LIN {X 0,Y 383.005,Z 334.275,A -85,B 0,C 180,E1 -11834.306,E2 -11834.306} C_VEL
LIN {X 0,Y 383.071,Z 334.265,A -85,B 0,C 180,E1 -11837.25,E2 -11837.25} C_VEL
LIN {X 0,Y 383.019,Z 334.272,A -85,B 0,C 180,E1 -11840.413,E2 -11840.413} C_VEL
LIN {X 0,Y 383.023,Z 334.273,A -85,B 0,C 180,E1 -11844.045,E2 -11844.045} C_VEL
LIN {X 0,Y 383.002,Z 334.279,A -85,B 0,C 180,E1 -11847.574,E2 -11847.574} C_VEL
LIN {X 0,Y 382.989,Z 334.275,A -85,B 0,C 180,E1 -11850.301,E2 -11850.301} C_VEL
LIN {X 0,Y 383.054,Z 334.267,A -85,B 0,C 180,E1 -11852.699,E2 -11852.699} C_VEL
LIN {X 0,Y 383.049,Z 334.27,A -85,B 0,C 180,E1 -11855.04,E2 -11855.04} C_VEL
LIN {X 0,Y 382.99,Z 334.275,A -85,B 0,C 180,E1 -11858.47,E2 -11858.47} C_VEL
LIN {X 0,Y 383.087,Z 334.264,A -85,B 0,C 180,E1 -11861.828,E2 -11861.828} C_VEL
LIN {X 0,Y 383.108,Z 334.266,A -85,B 0,C 180,E1 -11865.119,E2 -11865.119} C_VEL
LIN {X 0,Y 383.096,Z 334.262,A -85,B 0,C 180,E1 -11868.358,E2 -11868.358} C_VEL
LIN {X 0,Y 383.262,Z 334.241,A -85,B 0,C 180,E1 -11871.977,E2 -11871.977} C_VEL
LIN {X 0,Y 383.196,Z 334.253,A -85,B 0,C 180,E1 -11874.739,E2 -11874.739} C_VEL
LIN {X 0,Y 383.387,Z 334.225,A -85,B 0,C 180,E1 -11877.899,E2 -11877.899} C_VEL
LIN {X 0,Y 383.517,Z 334.209,A -85,B 0,C 180,E1 -11880.001,E2 -11880.001} C_VEL
LIN {X 0,Y 383.249,Z 334.245,A -85,B 0,C 180,E1 -11883.154,E2 -11883.154} C_VEL
LIN {X 0,Y 383.28,Z 334.241,A -85,B 0,C 180,E1 -11886.317,E2 -11886.317} C_VEL
LIN {X 0,Y 383.151,Z 334.254,A -85,B 0,C 180,E1 -11889.503,E2 -11889.503} C_VEL
LIN {X 0,Y 383.125,Z 334.258,A -85,B 0,C 180,E1 -11893.537,E2 -11893.537} C_VEL
LIN {X 0,Y 383.094,Z 334.262,A -85,B 0,C 180,E1 -11897.07,E2 -11897.07} C_VEL
LIN {X 0,Y 383.034,Z 334.272,A -85,B 0,C 180,E1 -11900.65,E2 -11900.65} C_VEL
LIN {X 0,Y 383.023,Z 334.272,A -85,B 0,C 180,E1 -11903.809,E2 -11903.809} C_VEL
LIN {X 0,Y 383.08,Z 334.269,A -85,B 0,C 180,E1 -11906.124,E2 -11906.124} C_VEL
LIN {X 0,Y 383.018,Z 334.274,A -85,B 0,C 180,E1 -11908.495,E2 -11908.495} C_VEL
LIN {X 0,Y 383.011,Z 334.277,A -85,B 0,C 180,E1 -11912.15,E2 -11912.15} C_VEL
LIN {X 0,Y 383.019,Z 334.275,A -85,B 0,C 180,E1 -11914.668,E2 -11914.668} C_VEL
LIN {X 0,Y 383.004,Z 334.279,A -85,B 0,C 180,E1 -11917.905,E2 -11917.905} C_VEL
LIN {X 0,Y 383.462,Z 337.13,A -85,B 0,C 180,E1 -11921.285,E2 -11921.285} C_VEL
LIN {X 0,Y 383.825,Z 340.043,A -85,B 0,C 180,E1 -11924.43,E2 -11924.43} C_VEL
LIN {X 0,Y 384.05,Z 343.012,A -85,B 0,C 180,E1 -11927.384,E2 -11927.384} C_VEL
LIN {X 0,Y 383.867,Z 346.172,A -85,B 0,C 180,E1 -11930.261,E2 -11930.261} C_VEL
LIN {X 0,Y 383.627,Z 349.135,A -85,B 0,C 180,E1 -11932.803,E2 -11932.803} C_VEL
LIN {X 0,Y 383.165,Z 353.821,A -85,B 0,C 180,E1 -11936.615,E2 -11936.615} C_VEL
LIN {X 0,Y 382.799,Z 357.743,A -85,B 0,C 180,E1 -11939.644,E2 -11939.644} C_VEL
LIN {X 0,Y 382.466,Z 361.805,A -85,B 0,C 180,E1 -11942.653,E2 -11942.653} C_VEL
LIN {X 0,Y 382.125,Z 366.674,A -85,B 0,C 180,E1 -11946.133,E2 -11946.133} C_VEL
LIN {X 0,Y 381.861,Z 371.985,A -85,B 0,C 180,E1 -11949.825,E2 -11949.825} C_VEL
LIN {X 0,Y 381.764,Z 373.941,A -85,B 0,C 180,E1 -11951.102,E2 -11951.102} C_VEL
LIN {X 0,Y 383.92,Z 384.326,A -85,B 0,C 180,E1 -11951.558,E2 -11951.558} C_VEL
LIN {X 0,Y 385.496,Z 393.257,A -85,B 0,C 180,E1 -11952.049,E2 -11952.049} C_VEL
LIN {X 0,Y 386.748,Z 402.194,A -85,B 0,C 180,E1 -11952.633,E2 -11952.633} C_VEL
LIN {X 0,Y 387.052,Z 408.906,A -85,B 0,C 180,E1 -11953.111,E2 -11953.111} C_VEL
LIN {X 0,Y 386.18,Z 419.818,A -85,B 0,C 180,E1 -11954.023,E2 -11954.023} C_VEL
LIN {X 0,Y 385.324,Z 428.762,A -85,B 0,C 180,E1 -11954.935,E2 -11954.935} C_VEL
LIN {X 0,Y 384.664,Z 436.503,A -85,B 0,C 180,E1 -11955.879,E2 -11955.879} C_VEL
LIN {X 0,Y 383.999,Z 444.518,A -85,B 0,C 180,E1 -11957.044,E2 -11957.044} C_VEL
LIN {X 0,Y 383.347,Z 450.719,A -85,B 0,C 180,E1 -11958.097,E2 -11958.097} C_VEL
LIN {X 0,Y 382.763,Z 457.257,A -85,B 0,C 180,E1 -11959.42,E2 -11959.42} C_VEL
LIN {X 0,Y 382.4,Z 461.76,A -85,B 0,C 180,E1 -11960.479,E2 -11960.479} C_VEL
LIN {X 0,Y 381.991,Z 467.252,A -85,B 0,C 180,E1 -11962.069,E2 -11962.069} C_VEL
LIN {X 0,Y 381.713,Z 471.576,A -85,B 0,C 180,E1 -11963.658,E2 -11963.658} C_VEL
LIN {X 0,Y 381.646,Z 473.944,A -85,B 0,C 180,E1 -11964.717,E2 -11964.717} C_VEL
LIN {X 0,Y 381.627,Z 475.743,A -85,B 0,C 180,E1 -11965.776,E2 -11965.776} C_VEL
LIN {X 0,Y 381.56,Z 478.187,A -85,B 0,C 180,E1 -11967.889,E2 -11967.889} C_VEL
LIN {X 0,Y 381.603,Z 478.776,A -85,B 0,C 180,E1 -11968.945,E2 -11968.945} C_VEL
LIN {X 0,Y 381.603,Z 478.776,A -85,B 0,C 180,E1 -11971.055,E2 -11971.055} C_VEL
LIN {X 0,Y 381.56,Z 478.187,A -85,B 0,C 180,E1 -11972.111,E2 -11972.111} C_VEL
LIN {X 0,Y 381.627,Z 475.743,A -85,B 0,C 180,E1 -11974.224,E2 -11974.224} C_VEL
LIN {X 0,Y 381.644,Z 473.943,A -85,B 0,C 180,E1 -11975.283,E2 -11975.283} C_VEL
LIN {X 0,Y 381.783,Z 470.336,A -85,B 0,C 180,E1 -11976.872,E2 -11976.872} C_VEL
LIN {X 0,Y 382.116,Z 465.592,A -85,B 0,C 180,E1 -11978.461,E2 -11978.461} C_VEL
LIN {X 0,Y 382.541,Z 459.568,A -85,B 0,C 180,E1 -11980.051,E2 -11980.051} C_VEL
LIN {X 0,Y 383.075,Z 453.471,A -85,B 0,C 180,E1 -11981.375,E2 -11981.375} C_VEL
LIN {X 0,Y 383.666,Z 447.771,A -85,B 0,C 180,E1 -11982.429,E2 -11982.429} C_VEL
LIN {X 0,Y 384.398,Z 439.214,A -85,B 0,C 180,E1 -11983.75,E2 -11983.75} C_VEL
LIN {X 0,Y 385.098,Z 431.032,A -85,B 0,C 180,E1 -11984.803,E2 -11984.803} C_VEL
LIN {X 0,Y 385.884,Z 422.52,A -85,B 0,C 180,E1 -11985.719,E2 -11985.719} C_VEL
LIN {X 0,Y 386.66,Z 413.804,A -85,B 0,C 180,E1 -11986.499,E2 -11986.499} C_VEL
LIN {X 0,Y 387.148,Z 406.33,A -85,B 0,C 180,E1 -11987.07,E2 -11987.07} C_VEL
LIN {X 0,Y 385.973,Z 396.427,A -85,B 0,C 180,E1 -11987.761,E2 -11987.761} C_VEL
LIN {X 0,Y 384.121,Z 385.213,A -85,B 0,C 180,E1 -11988.397,E2 -11988.397} C_VEL
LIN {X 0,Y 381.855,Z 374.444,A -85,B 0,C 180,E1 -11988.88,E2 -11988.88} C_VEL
LIN {X 0,Y 381.785,Z 373.753,A -85,B 0,C 180,E1 -11988.931,E2 -11988.931} C_VEL
LIN {X 0,Y 381.957,Z 369.9,A -85,B 0,C 180,E1 -11991.592,E2 -11991.592} C_VEL
LIN {X 0,Y 382.246,Z 365.004,A -85,B 0,C 180,E1 -11995.016,E2 -11995.016} C_VEL
LIN {X 0,Y 382.585,Z 360.178,A -85,B 0,C 180,E1 -11998.53,E2 -11998.53} C_VEL
LIN {X 0,Y 383.044,Z 355.398,A -85,B 0,C 180,E1 -12002.146,E2 -12002.146} C_VEL
LIN {X 0,Y 383.447,Z 350.679,A -85,B 0,C 180,E1 -12005.91,E2 -12005.91} C_VEL
LIN {X 0,Y 383.765,Z 347.567,A -85,B 0,C 180,E1 -12008.51,E2 -12008.51} C_VEL
LIN {X 0,Y 383.998,Z 344.341,A -85,B 0,C 180,E1 -12011.375,E2 -12011.375} C_VEL
LIN {X 0,Y 383.996,Z 341.509,A -85,B 0,C 180,E1 -12014.066,E2 -12014.066} C_VEL
LIN {X 0,Y 383.581,Z 338.384,A -85,B 0,C 180,E1 -12017.318,E2 -12017.318} C_VEL
LIN {X 0,Y 383.229,Z 335.695,A -85,B 0,C 180,E1 -12020.374,E2 -12020.374} C_VEL
LIN {X 0,Y 383.004,Z 334.279,A -85,B 0,C 180,E1 -12022.095,E2 -12022.095} C_VEL
LIN {X 0,Y 383.019,Z 334.278,A -85,B 0,C 180,E1 -12025.332,E2 -12025.332} C_VEL
LIN {X 0,Y 382.984,Z 334.275,A -85,B 0,C 180,E1 -12029.081,E2 -12029.081} C_VEL
LIN {X 0,Y 383.057,Z 334.266,A -85,B 0,C 180,E1 -12032.698,E2 -12032.698} C_VEL
LIN {X 0,Y 383.051,Z 334.267,A -85,B 0,C 180,E1 -12035.039,E2 -12035.039} C_VEL
LIN {X 0,Y 382.995,Z 334.274,A -85,B 0,C 180,E1 -12038.469,E2 -12038.469} C_VEL
LIN {X 0,Y 383.053,Z 334.271,A -85,B 0,C 180,E1 -12041.825,E2 -12041.825} C_VEL
LIN {X 0,Y 383.11,Z 334.262,A -85,B 0,C 180,E1 -12045.118,E2 -12045.118} C_VEL
LIN {X 0,Y 383.097,Z 334.261,A -85,B 0,C 180,E1 -12048.357,E2 -12048.357} C_VEL
LIN {X 0,Y 383.263,Z 334.241,A -85,B 0,C 180,E1 -12051.975,E2 -12051.975} C_VEL
LIN {X 0,Y 383.196,Z 334.25,A -85,B 0,C 180,E1 -12054.738,E2 -12054.738} C_VEL
LIN {X 0,Y 383.387,Z 334.226,A -85,B 0,C 180,E1 -12057.898,E2 -12057.898} C_VEL
LIN {X 0,Y 383.517,Z 334.209,A -85,B 0,C 180,E1 -12059.999,E2 -12059.999} C_VEL
LIN {X 0,Y 383.25,Z 334.248,A -85,B 0,C 180,E1 -12063.153,E2 -12063.153} C_VEL
LIN {X 0,Y 383.262,Z 334.24,A -85,B 0,C 180,E1 -12066.542,E2 -12066.542} C_VEL
LIN {X 0,Y 383.15,Z 334.256,A -85,B 0,C 180,E1 -12069.502,E2 -12069.502} C_VEL
LIN {X 0,Y 383.123,Z 334.258,A -85,B 0,C 180,E1 -12073.536,E2 -12073.536} C_VEL
LIN {X 0,Y 383.093,Z 334.262,A -85,B 0,C 180,E1 -12077.454,E2 -12077.454} C_VEL
LIN {X 0,Y 383.027,Z 334.276,A -85,B 0,C 180,E1 -12080.646,E2 -12080.646} C_VEL
LIN {X 0,Y 383.023,Z 334.271,A -85,B 0,C 180,E1 -12083.807,E2 -12083.807} C_VEL
LIN {X 0,Y 383.077,Z 334.266,A -85,B 0,C 180,E1 -12086.123,E2 -12086.123} C_VEL
LIN {X 0,Y 383.037,Z 334.275,A -85,B 0,C 180,E1 -12088.492,E2 -12088.492} C_VEL
LIN {X 0,Y 383.006,Z 334.276,A -85,B 0,C 180,E1 -12092.149,E2 -12092.149} C_VEL
LIN {X 0,Y 383.015,Z 334.274,A -85,B 0,C 180,E1 -12094.667,E2 -12094.667} C_VEL
LIN {X 0,Y 383,Z 334.276,A -85,B 0,C 180,E1 -12097.904,E2 -12097.904} C_VEL
LIN {X 0,Y 383.043,Z 334.268,A -85,B 0,C 180,E1 -12101.339,E2 -12101.339} C_VEL
LIN {X 0,Y 383.033,Z 334.273,A -85,B 0,C 180,E1 -12104.309,E2 -12104.309} C_VEL
LIN {X 0,Y 383.036,Z 334.269,A -85,B 0,C 180,E1 -12107.244,E2 -12107.244} C_VEL
LIN {X 0,Y 383.018,Z 334.273,A -85,B 0,C 180,E1 -12110.412,E2 -12110.412} C_VEL
LIN {X 0,Y 383.023,Z 334.275,A -85,B 0,C 180,E1 -12114.044,E2 -12114.044} C_VEL
LIN {X 0,Y 382.983,Z 334.28,A -85,B 0,C 180,E1 -12117.578,E2 -12117.578} C_VEL
LIN {X 0,Y 382.988,Z 334.276,A -85,B 0,C 180,E1 -12120.3,E2 -12120.3} C_VEL
LIN {X 0,Y 383.053,Z 334.267,A -85,B 0,C 180,E1 -12122.698,E2 -12122.698} C_VEL
LIN {X 0,Y 383.03,Z 334.27,A -85,B 0,C 180,E1 -12126.193,E2 -12126.193} C_VEL
LIN {X 0,Y 383.056,Z 334.272,A -85,B 0,C 180,E1 -12129.599,E2 -12129.599} C_VEL
LIN {X 0,Y 383.101,Z 334.266,A -85,B 0,C 180,E1 -12132.931,E2 -12132.931} C_VEL
LIN {X 0,Y 383.121,Z 334.263,A -85,B 0,C 180,E1 -12136.464,E2 -12136.464} C_VEL
LIN {X 0,Y 383.139,Z 334.266,A -85,B 0,C 180,E1 -12139.597,E2 -12139.597} C_VEL
LIN {X 0,Y 383.738,Z 336.384,A -85,B 0,C 180,E1 -12139.914,E2 -12139.914} C_VEL
LIN {X 0,Y 385.2,Z 338.424,A -85,B 0,C 180,E1 -12140.615,E2 -12140.615} C_VEL
LIN {X 0,Y 387.437,Z 339.864,A -85,B 0,C 180,E1 -12141.656,E2 -12141.656} C_VEL
LIN {X 0,Y 388.84,Z 340.559,A -85,B 0,C 180,E1 -12142.402,E2 -12142.402} C_VEL
LIN {X 0,Y 389.961,Z 342.834,A -85,B 0,C 180,E1 -12143.142,E2 -12143.142} C_VEL
LIN {X 0,Y 391.789,Z 344.996,A -85,B 0,C 180,E1 -12144.467,E2 -12144.467} C_VEL
LIN {X 0,Y 393.422,Z 346.061,A -85,B 0,C 180,E1 -12145.902,E2 -12145.902} C_VEL
LIN {X 0,Y 394.945,Z 346.431,A -85,B 0,C 180,E1 -12147.96,E2 -12147.96} C_VEL
LIN {X 0,Y 395.509,Z 346.494,A -85,B 0,C 180,E1 -12150,E2 -12150} C_VEL
LIN {X 0,Y 394.945,Z 346.431,A -85,B 0,C 180,E1 -12152.04,E2 -12152.04} C_VEL
LIN {X 0,Y 393.422,Z 346.062,A -85,B 0,C 180,E1 -12154.098,E2 -12154.098} C_VEL
LIN {X 0,Y 391.445,Z 344.701,A -85,B 0,C 180,E1 -12155.796,E2 -12155.796} C_VEL
LIN {X 0,Y 389.552,Z 342.156,A -85,B 0,C 180,E1 -12157.135,E2 -12157.135} C_VEL
LIN {X 0,Y 388.788,Z 340.393,A -85,B 0,C 180,E1 -12157.634,E2 -12157.634} C_VEL
LIN {X 0,Y 385.957,Z 339.051,A -85,B 0,C 180,E1 -12159.036,E2 -12159.036} C_VEL
LIN {X 0,Y 384.054,Z 336.971,A -85,B 0,C 180,E1 -12159.938,E2 -12159.938} C_VEL
LIN {X 0,Y 383.252,Z 334.909,A -85,B 0,C 180,E1 -12160.333,E2 -12160.333} C_VEL
LIN {X 0,Y 383.121,Z 334.263,A -85,B 0,C 180,E1 -12160.436,E2 -12160.436} C_VEL
LIN {X 0,Y 383.123,Z 334.262,A -85,B 0,C 180,E1 -12163.796,E2 -12163.796} C_VEL
LIN {X 0,Y 383.091,Z 334.266,A -85,B 0,C 180,E1 -12167.455,E2 -12167.455} C_VEL
LIN {X 0,Y 383.03,Z 334.274,A -85,B 0,C 180,E1 -12170.649,E2 -12170.649} C_VEL
LIN {X 0,Y 383.03,Z 334.27,A -85,B 0,C 180,E1 -12173.807,E2 -12173.807} C_VEL
LIN {X 0,Y 383.053,Z 334.267,A -85,B 0,C 180,E1 -12177.302,E2 -12177.302} C_VEL
LIN {X 0,Y 382.979,Z 334.277,A -85,B 0,C 180,E1 -12180.919,E2 -12180.919} C_VEL
LIN {X 0,Y 383.014,Z 334.273,A -85,B 0,C 180,E1 -12184.668,E2 -12184.668} C_VEL
LIN {X 0,Y 382.995,Z 334.274,A -85,B 0,C 180,E1 -12185.364,E2 -12185.364} C_VEL
LIN {X 0,Y 382.354,Z 334.359,A -85,B 0,C 180,E1 -12186.242,E2 -12186.242} C_VEL
LIN {X 0,Y 379.547,Z 334.716,A -85,B 0,C 180,E1 -12187.67,E2 -12187.67} C_VEL
LIN {X 0,Y 377.144,Z 335.017,A -85,B 0,C 180,E1 -12188.824,E2 -12188.824} C_VEL
LIN {X 0,Y 376.089,Z 335.143,A -85,B 0,C 180,E1 -12189.716,E2 -12189.716} C_VEL
LIN {X 0,Y 375.991,Z 335.152,A -85,B 0,C 180,E1 -12190.019,E2 -12190.019} C_VEL
LIN {X 0,Y 375.943,Z 335.157,A -85,B 0,C 180,E1 -12193.764,E2 -12193.764} C_VEL
LIN {X 0,Y 375.986,Z 335.147,A -85,B 0,C 180,E1 -12196.802,E2 -12196.802} C_VEL
LIN {X 0,Y 375.996,Z 335.15,A -85,B 0,C 180,E1 -12200.028,E2 -12200.028} C_VEL
LIN {X 0,Y 375.962,Z 335.154,A -85,B 0,C 180,E1 -12203.496,E2 -12203.496} C_VEL
LIN {X 0,Y 375.957,Z 335.154,A -85,B 0,C 180,E1 -12205.889,E2 -12205.889} C_VEL
LIN {X 0,Y 375.961,Z 335.155,A -85,B 0,C 180,E1 -12209.688,E2 -12209.688} C_VEL
LIN {X 0,Y 375.993,Z 335.147,A -85,B 0,C 180,E1 -12212.142,E2 -12212.142} C_VEL
LIN {X 0,Y 376.003,Z 335.145,A -85,B 0,C 180,E1 -12214.539,E2 -12214.539} C_VEL
LIN {X 0,Y 375.956,Z 335.151,A -85,B 0,C 180,E1 -12218.046,E2 -12218.046} C_VEL
LIN {X 0,Y 376.022,Z 335.147,A -85,B 0,C 180,E1 -12221.475,E2 -12221.475} C_VEL
LIN {X 0,Y 376.056,Z 335.141,A -85,B 0,C 180,E1 -12224.833,E2 -12224.833} C_VEL
LIN {X 0,Y 376.048,Z 335.139,A -85,B 0,C 180,E1 -12228.137,E2 -12228.137} C_VEL
LIN {X 0,Y 376.217,Z 335.118,A -85,B 0,C 180,E1 -12231.92,E2 -12231.92} C_VEL
LIN {X 0,Y 376.168,Z 335.127,A -85,B 0,C 180,E1 -12234.64,E2 -12234.64} C_VEL
LIN {X 0,Y 376.353,Z 335.101,A -85,B 0,C 180,E1 -12237.86,E2 -12237.86} C_VEL
LIN {X 0,Y 376.486,Z 335.085,A -85,B 0,C 180,E1 -12240.001,E2 -12240.001} C_VEL
LIN {X 0,Y 376.187,Z 335.124,A -85,B 0,C 180,E1 -12243.213,E2 -12243.213} C_VEL
LIN {X 0,Y 376.238,Z 335.12,A -85,B 0,C 180,E1 -12246.436,E2 -12246.436} C_VEL
LIN {X 0,Y 376.119,Z 335.13,A -85,B 0,C 180,E1 -12249.682,E2 -12249.682} C_VEL
LIN {X 0,Y 376.089,Z 335.134,A -85,B 0,C 180,E1 -12253.658,E2 -12253.658} C_VEL
LIN {X 0,Y 376.032,Z 335.141,A -85,B 0,C 180,E1 -12257.4,E2 -12257.4} C_VEL
LIN {X 0,Y 375.978,Z 335.149,A -85,B 0,C 180,E1 -12260.833,E2 -12260.833} C_VEL
LIN {X 0,Y 375.988,Z 335.153,A -85,B 0,C 180,E1 -12264.282,E2 -12264.282} C_VEL
LIN {X 0,Y 376.02,Z 335.145,A -85,B 0,C 180,E1 -12266.653,E2 -12266.653} C_VEL
LIN {X 0,Y 375.965,Z 335.154,A -85,B 0,C 180,E1 -12270.313,E2 -12270.313} C_VEL
LIN {X 0,Y 375.961,Z 335.157,A -85,B 0,C 180,E1 -12274.112,E2 -12274.112} C_VEL
LIN {X 0,Y 375.955,Z 335.156,A -85,B 0,C 180,E1 -12276.742,E2 -12276.742} C_VEL
LIN {X 0,Y 376.033,Z 335.725,A -85,B 0,C 180,E1 -12278.282,E2 -12278.282} C_VEL
LIN {X 0,Y 376.483,Z 338.576,A -85,B 0,C 180,E1 -12281.695,E2 -12281.695} C_VEL
LIN {X 0,Y 376.879,Z 341.755,A -85,B 0,C 180,E1 -12285.123,E2 -12285.123} C_VEL
LIN {X 0,Y 376.982,Z 344.5,A -85,B 0,C 180,E1 -12287.845,E2 -12287.845} C_VEL
LIN {X 0,Y 376.792,Z 347.545,A -85,B 0,C 180,E1 -12290.641,E2 -12290.641} C_VEL
LIN {X 0,Y 376.515,Z 350.697,A -85,B 0,C 180,E1 -12293.383,E2 -12293.383} C_VEL
LIN {X 0,Y 376.027,Z 355.41,A -85,B 0,C 180,E1 -12297.253,E2 -12297.253} C_VEL
LIN {X 0,Y 375.744,Z 358.488,A -85,B 0,C 180,E1 -12299.668,E2 -12299.668} C_VEL
LIN {X 0,Y 375.313,Z 363.296,A -85,B 0,C 180,E1 -12303.294,E2 -12303.294} C_VEL
LIN {X 0,Y 375.014,Z 368.142,A -85,B 0,C 180,E1 -12306.824,E2 -12306.824} C_VEL
LIN {X 0,Y 374.741,Z 373.736,A -85,B 0,C 180,E1 -12310.734,E2 -12310.734} C_VEL
LIN {X 0,Y 376.765,Z 383.476,A -85,B 0,C 180,E1 -12311.169,E2 -12311.169} C_VEL
LIN {X 0,Y 378.478,Z 393.112,A -85,B 0,C 180,E1 -12311.708,E2 -12311.708} C_VEL
LIN {X 0,Y 379.829,Z 402.363,A -85,B 0,C 180,E1 -12312.332,E2 -12312.332} C_VEL
LIN {X 0,Y 380.242,Z 408.71,A -85,B 0,C 180,E1 -12312.799,E2 -12312.799} C_VEL
LIN {X 0,Y 379.337,Z 419.622,A -85,B 0,C 180,E1 -12313.727,E2 -12313.727} C_VEL
LIN {X 0,Y 378.449,Z 428.566,A -85,B 0,C 180,E1 -12314.655,E2 -12314.655} C_VEL
LIN {X 0,Y 377.606,Z 437.835,A -85,B 0,C 180,E1 -12315.829,E2 -12315.829} C_VEL
LIN {X 0,Y 376.887,Z 445.948,A -85,B 0,C 180,E1 -12317.07,E2 -12317.07} C_VEL
LIN {X 0,Y 376.219,Z 451.898,A -85,B 0,C 180,E1 -12318.142,E2 -12318.142} C_VEL
LIN {X 0,Y 375.658,Z 458.217,A -85,B 0,C 180,E1 -12319.49,E2 -12319.49} C_VEL
LIN {X 0,Y 375.215,Z 463.48,A -85,B 0,C 180,E1 -12320.839,E2 -12320.839} C_VEL
LIN {X 0,Y 374.809,Z 468.609,A -85,B 0,C 180,E1 -12322.458,E2 -12322.458} C_VEL
LIN {X 0,Y 374.586,Z 472.267,A -85,B 0,C 180,E1 -12323.931,E2 -12323.931} C_VEL
LIN {X 0,Y 374.553,Z 475.547,A -85,B 0,C 180,E1 -12325.696,E2 -12325.696} C_VEL
LIN {X 0,Y 374.459,Z 477.991,A -85,B 0,C 180,E1 -12327.849,E2 -12327.849} C_VEL
LIN {X 0,Y 374.503,Z 478.581,A -85,B 0,C 180,E1 -12328.925,E2 -12328.925} C_VEL
LIN {X 0,Y 374.503,Z 478.581,A -85,B 0,C 180,E1 -12331.075,E2 -12331.075} C_VEL
LIN {X 0,Y 374.459,Z 477.991,A -85,B 0,C 180,E1 -12332.151,E2 -12332.151} C_VEL
LIN {X 0,Y 374.553,Z 475.547,A -85,B 0,C 180,E1 -12334.304,E2 -12334.304} C_VEL
LIN {X 0,Y 374.584,Z 472.274,A -85,B 0,C 180,E1 -12336.066,E2 -12336.066} C_VEL
LIN {X 0,Y 374.809,Z 468.609,A -85,B 0,C 180,E1 -12337.542,E2 -12337.542} C_VEL
LIN {X 0,Y 375.215,Z 463.48,A -85,B 0,C 180,E1 -12339.161,E2 -12339.161} C_VEL
LIN {X 0,Y 375.657,Z 458.217,A -85,B 0,C 180,E1 -12340.51,E2 -12340.51} C_VEL
LIN {X 0,Y 376.221,Z 451.898,A -85,B 0,C 180,E1 -12341.858,E2 -12341.858} C_VEL
LIN {X 0,Y 376.888,Z 445.948,A -85,B 0,C 180,E1 -12342.93,E2 -12342.93} C_VEL
LIN {X 0,Y 377.606,Z 437.829,A -85,B 0,C 180,E1 -12344.172,E2 -12344.172} C_VEL
LIN {X 0,Y 378.312,Z 429.7,A -85,B 0,C 180,E1 -12345.213,E2 -12345.213} C_VEL
LIN {X 0,Y 379.163,Z 420.972,A -85,B 0,C 180,E1 -12346.143,E2 -12346.143} C_VEL
LIN {X 0,Y 379.955,Z 411.975,A -85,B 0,C 180,E1 -12346.937,E2 -12346.937} C_VEL
LIN {X 0,Y 380.215,Z 406.272,A -85,B 0,C 180,E1 -12347.382,E2 -12347.382} C_VEL
LIN {X 0,Y 378.828,Z 395.108,A -85,B 0,C 180,E1 -12348.167,E2 -12348.167} C_VEL
LIN {X 0,Y 376.872,Z 384.021,A -85,B 0,C 180,E1 -12348.803,E2 -12348.803} C_VEL
LIN {X 0,Y 374.76,Z 373.587,A -85,B 0,C 180,E1 -12349.3,E2 -12349.3} C_VEL
LIN {X 0,Y 375.022,Z 367.931,A -85,B 0,C 180,E1 -12353.324,E2 -12353.324} C_VEL
LIN {X 0,Y 375.314,Z 363.287,A -85,B 0,C 180,E1 -12356.706,E2 -12356.706} C_VEL
LIN {X 0,Y 375.745,Z 358.481,A -85,B 0,C 180,E1 -12360.332,E2 -12360.332} C_VEL
LIN {X 0,Y 376.172,Z 353.737,A -85,B 0,C 180,E1 -12364.089,E2 -12364.089} C_VEL
LIN {X 0,Y 376.66,Z 349.076,A -85,B 0,C 180,E1 -12368.005,E2 -12368.005} C_VEL
LIN {X 0,Y 376.915,Z 346.003,A -85,B 0,C 180,E1 -12370.739,E2 -12370.739} C_VEL
LIN {X 0,Y 376.992,Z 342.998,A -85,B 0,C 180,E1 -12373.611,E2 -12373.611} C_VEL
LIN {X 0,Y 376.651,Z 340.041,A -85,B 0,C 180,E1 -12376.694,E2 -12376.694} C_VEL
LIN {X 0,Y 376.265,Z 337.155,A -85,B 0,C 180,E1 -12379.979,E2 -12379.979} C_VEL
LIN {X 0,Y 376.012,Z 335.567,A -85,B 0,C 180,E1 -12381.917,E2 -12381.917} C_VEL
LIN {X 0,Y 375.965,Z 335.155,A -85,B 0,C 180,E1 -12383.495,E2 -12383.495} C_VEL
LIN {X 0,Y 375.961,Z 335.157,A -85,B 0,C 180,E1 -12385.888,E2 -12385.888} C_VEL
LIN {X 0,Y 375.965,Z 335.154,A -85,B 0,C 180,E1 -12389.687,E2 -12389.687} C_VEL
LIN {X 0,Y 376.02,Z 335.145,A -85,B 0,C 180,E1 -12393.347,E2 -12393.347} C_VEL
LIN {X 0,Y 375.979,Z 335.148,A -85,B 0,C 180,E1 -12396.887,E2 -12396.887} C_VEL
LIN {X 0,Y 375.999,Z 335.146,A -85,B 0,C 180,E1 -12400.339,E2 -12400.339} C_VEL
LIN {X 0,Y 376.026,Z 335.147,A -85,B 0,C 180,E1 -12403.718,E2 -12403.718} C_VEL
LIN {X 0,Y 376.103,Z 335.134,A -85,B 0,C 180,E1 -12407.041,E2 -12407.041} C_VEL
LIN {X 0,Y 376.119,Z 335.13,A -85,B 0,C 180,E1 -12410.318,E2 -12410.318} C_VEL
LIN {X 0,Y 376.238,Z 335.12,A -85,B 0,C 180,E1 -12413.564,E2 -12413.564} C_VEL
LIN {X 0,Y 376.353,Z 335.102,A -85,B 0,C 180,E1 -12417.859,E2 -12417.859} C_VEL
LIN {X 0,Y 376.486,Z 335.085,A -85,B 0,C 180,E1 -12419.999,E2 -12419.999} C_VEL
LIN {X 0,Y 376.188,Z 335.127,A -85,B 0,C 180,E1 -12423.212,E2 -12423.212} C_VEL
LIN {X 0,Y 376.229,Z 335.117,A -85,B 0,C 180,E1 -12426.529,E2 -12426.529} C_VEL
LIN {X 0,Y 376.118,Z 335.131,A -85,B 0,C 180,E1 -12429.681,E2 -12429.681} C_VEL
LIN {X 0,Y 376.088,Z 335.135,A -85,B 0,C 180,E1 -12433.657,E2 -12433.657} C_VEL
LIN {X 0,Y 376.042,Z 335.14,A -85,B 0,C 180,E1 -12437.607,E2 -12437.607} C_VEL
LIN {X 0,Y 375.976,Z 335.153,A -85,B 0,C 180,E1 -12440.832,E2 -12440.832} C_VEL
LIN {X 0,Y 375.987,Z 335.15,A -85,B 0,C 180,E1 -12444.281,E2 -12444.281} C_VEL
LIN {X 0,Y 376.017,Z 335.148,A -85,B 0,C 180,E1 -12446.652,E2 -12446.652} C_VEL
LIN {X 0,Y 375.967,Z 335.15,A -85,B 0,C 180,E1 -12449.079,E2 -12449.079} C_VEL
LIN {X 0,Y 375.953,Z 335.153,A -85,B 0,C 180,E1 -12452.827,E2 -12452.827} C_VEL
LIN {X 0,Y 375.955,Z 335.151,A -85,B 0,C 180,E1 -12455.415,E2 -12455.415} C_VEL
LIN {X 0,Y 375.974,Z 335.155,A -85,B 0,C 180,E1 -12458.271,E2 -12458.271} C_VEL
LIN {X 0,Y 375.986,Z 335.148,A -85,B 0,C 180,E1 -12461.61,E2 -12461.61} C_VEL
LIN {X 0,Y 375.967,Z 335.15,A -85,B 0,C 180,E1 -12465.262,E2 -12465.262} C_VEL
LIN {X 0,Y 375.977,Z 335.148,A -85,B 0,C 180,E1 -12469.138,E2 -12469.138} C_VEL
LIN {X 0,Y 375.964,Z 335.156,A -85,B 0,C 180,E1 -12471.912,E2 -12471.912} C_VEL
LIN {X 0,Y 375.976,Z 335.15,A -85,B 0,C 180,E1 -12475.332,E2 -12475.332} C_VEL
LIN {X 0,Y 375.954,Z 335.152,A -85,B 0,C 180,E1 -12478.438,E2 -12478.438} C_VEL
LIN {X 0,Y 375.992,Z 335.148,A -85,B 0,C 180,E1 -12482.141,E2 -12482.141} C_VEL
LIN {X 0,Y 376.002,Z 335.145,A -85,B 0,C 180,E1 -12484.539,E2 -12484.539} C_VEL
LIN {X 0,Y 375.961,Z 335.152,A -85,B 0,C 180,E1 -12488.046,E2 -12488.046} C_VEL
LIN {X 0,Y 376.021,Z 335.149,A -85,B 0,C 180,E1 -12491.474,E2 -12491.474} C_VEL
LIN {X 0,Y 376.055,Z 335.144,A -85,B 0,C 180,E1 -12494.833,E2 -12494.833} C_VEL
LIN {X 0,Y 376.117,Z 335.308,A -85,B 0,C 180,E1 -12497.317,E2 -12497.317} C_VEL
LIN {X 0,Y 376.775,Z 337.476,A -85,B 0,C 180,E1 -12497.613,E2 -12497.613} C_VEL
LIN {X 0,Y 378.603,Z 339.764,A -85,B 0,C 180,E1 -12498.286,E2 -12498.286} C_VEL
LIN {X 0,Y 381.129,Z 341.2,A -85,B 0,C 180,E1 -12499.206,E2 -12499.206} C_VEL
LIN {X 0,Y 382.563,Z 343.884,A -85,B 0,C 180,E1 -12499.849,E2 -12499.849} C_VEL
LIN {X 0,Y 384.983,Z 346.162,A -85,B 0,C 180,E1 -12500.941,E2 -12500.941} C_VEL
LIN {X 0,Y 387.406,Z 347.441,A -85,B 0,C 180,E1 -12502.125,E2 -12502.125} C_VEL
LIN {X 0,Y 388.935,Z 349.999,A -85,B 0,C 180,E1 -12503.079,E2 -12503.079} C_VEL
LIN {X 0,Y 390.889,Z 352.078,A -85,B 0,C 180,E1 -12504.454,E2 -12504.454} C_VEL
LIN {X 0,Y 392.534,Z 353.091,A -85,B 0,C 180,E1 -12505.893,E2 -12505.893} C_VEL
LIN {X 0,Y 394.083,Z 353.478,A -85,B 0,C 180,E1 -12507.956,E2 -12507.956} C_VEL
LIN {X 0,Y 394.645,Z 353.533,A -85,B 0,C 180,E1 -12510,E2 -12510} C_VEL
LIN {X 0,Y 394.082,Z 353.477,A -85,B 0,C 180,E1 -12512.044,E2 -12512.044} C_VEL
LIN {X 0,Y 392.534,Z 353.092,A -85,B 0,C 180,E1 -12514.107,E2 -12514.107} C_VEL
LIN {X 0,Y 390.528,Z 351.798,A -85,B 0,C 180,E1 -12515.81,E2 -12515.81} C_VEL
LIN {X 0,Y 388.395,Z 349.209,A -85,B 0,C 180,E1 -12517.277,E2 -12517.277} C_VEL
LIN {X 0,Y 387.179,Z 347.137,A -85,B 0,C 180,E1 -12518.008,E2 -12518.008} C_VEL
LIN {X 0,Y 384.526,Z 345.833,A -85,B 0,C 180,E1 -12519.267,E2 -12519.267} C_VEL
LIN {X 0,Y 382.398,Z 343.659,A -85,B 0,C 180,E1 -12520.222,E2 -12520.222} C_VEL
LIN {X 0,Y 380.993,Z 341.031,A -85,B 0,C 180,E1 -12520.852,E2 -12520.852} C_VEL
LIN {X 0,Y 378.582,Z 339.746,A -85,B 0,C 180,E1 -12521.722,E2 -12521.722} C_VEL
LIN {X 0,Y 376.775,Z 337.476,A -85,B 0,C 180,E1 -12522.387,E2 -12522.387} C_VEL
LIN {X 0,Y 376.109,Z 335.138,A -85,B 0,C 180,E1 -12522.718,E2 -12522.718} C_VEL
LIN {X 0,Y 376.025,Z 335.147,A -85,B 0,C 180,E1 -12526.281,E2 -12526.281} C_VEL
LIN {X 0,Y 375.996,Z 335.148,A -85,B 0,C 180,E1 -12529.661,E2 -12529.661} C_VEL
LIN {X 0,Y 375.992,Z 335.147,A -85,B 0,C 180,E1 -12533.668,E2 -12533.668} C_VEL
LIN {X 0,Y 376.016,Z 335.147,A -85,B 0,C 180,E1 -12536.652,E2 -12536.652} C_VEL
LIN {X 0,Y 375.966,Z 335.15,A -85,B 0,C 180,E1 -12539.079,E2 -12539.079} C_VEL
LIN {X 0,Y 375.947,Z 335.153,A -85,B 0,C 180,E1 -12542.829,E2 -12542.829} C_VEL
LIN {X 0,Y 375.955,Z 335.151,A -85,B 0,C 180,E1 -12545.416,E2 -12545.416} C_VEL
LIN {X 0,Y 375.974,Z 335.153,A -85,B 0,C 180,E1 -12548.271,E2 -12548.271} C_VEL
LIN {X 0,Y 375.991,Z 335.152,A -85,B 0,C 180,E1 -12550.019,E2 -12550.019} C_VEL
LIN {X 0,Y 375.278,Z 335.235,A -85,B 0,C 180,E1 -12550.912,E2 -12550.912} C_VEL
LIN {X 0,Y 372.374,Z 335.599,A -85,B 0,C 180,E1 -12552.364,E2 -12552.364} C_VEL
LIN {X 0,Y 369.966,Z 335.899,A -85,B 0,C 180,E1 -12553.539,E2 -12553.539} C_VEL
LIN {X 0,Y 368.975,Z 336.022,A -85,B 0,C 180,E1 -12554.447,E2 -12554.447} C_VEL
LIN {X 0,Y 368.916,Z 336.027,A -85,B 0,C 180,E1 -12554.755,E2 -12554.755} C_VEL
LIN {X 0,Y 368.942,Z 336.027,A -85,B 0,C 180,E1 -12558.187,E2 -12558.187} C_VEL
LIN {X 0,Y 368.909,Z 336.031,A -85,B 0,C 180,E1 -12561.359,E2 -12561.359} C_VEL
LIN {X 0,Y 368.933,Z 336.027,A -85,B 0,C 180,E1 -12565.147,E2 -12565.147} C_VEL
LIN {X 0,Y 368.926,Z 336.028,A -85,B 0,C 180,E1 -12569.047,E2 -12569.047} C_VEL
LIN {X 0,Y 368.977,Z 336.026,A -85,B 0,C 180,E1 -12571.564,E2 -12571.564} C_VEL
LIN {X 0,Y 368.997,Z 336.019,A -85,B 0,C 180,E1 -12574.02,E2 -12574.02} C_VEL
LIN {X 0,Y 368.923,Z 336.031,A -85,B 0,C 180,E1 -12577.605,E2 -12577.605} C_VEL
LIN {X 0,Y 368.98,Z 336.024,A -85,B 0,C 180,E1 -12581.108,E2 -12581.108} C_VEL
LIN {X 0,Y 368.996,Z 336.018,A -85,B 0,C 180,E1 -12584.536,E2 -12584.536} C_VEL
LIN {X 0,Y 369.003,Z 336.017,A -85,B 0,C 180,E1 -12587.907,E2 -12587.907} C_VEL
LIN {X 0,Y 369.186,Z 335.994,A -85,B 0,C 180,E1 -12591.847,E2 -12591.847} C_VEL
LIN {X 0,Y 369.141,Z 336.002,A -85,B 0,C 180,E1 -12594.538,E2 -12594.538} C_VEL
LIN {X 0,Y 369.318,Z 335.978,A -85,B 0,C 180,E1 -12597.819,E2 -12597.819} C_VEL
LIN {X 0,Y 369.456,Z 335.961,A -85,B 0,C 180,E1 -12600.001,E2 -12600.001} C_VEL
LIN {X 0,Y 369.318,Z 335.979,A -85,B 0,C 180,E1 -12602.182,E2 -12602.182} C_VEL
LIN {X 0,Y 369.198,Z 335.998,A -85,B 0,C 180,E1 -12606.559,E2 -12606.559} C_VEL
LIN {X 0,Y 369.121,Z 336.007,A -85,B 0,C 180,E1 -12608.762,E2 -12608.762} C_VEL
LIN {X 0,Y 369.005,Z 336.019,A -85,B 0,C 180,E1 -12612.094,E2 -12612.094} C_VEL
LIN {X 0,Y 368.997,Z 336.018,A -85,B 0,C 180,E1 -12615.465,E2 -12615.465} C_VEL
LIN {X 0,Y 368.955,Z 336.024,A -85,B 0,C 180,E1 -12618.895,E2 -12618.895} C_VEL
LIN {X 0,Y 368.924,Z 336.032,A -85,B 0,C 180,E1 -12622.396,E2 -12622.396} C_VEL
LIN {X 0,Y 369,Z 336.021,A -85,B 0,C 180,E1 -12625.981,E2 -12625.981} C_VEL
LIN {X 0,Y 368.915,Z 336.03,A -85,B 0,C 180,E1 -12629.691,E2 -12629.691} C_VEL
LIN {X 0,Y 368.898,Z 336.03,A -85,B 0,C 180,E1 -12633.044,E2 -12633.044} C_VEL
LIN {X 0,Y 368.918,Z 336.034,A -85,B 0,C 180,E1 -12636.197,E2 -12636.197} C_VEL
LIN {X 0,Y 368.946,Z 336.298,A -85,B 0,C 180,E1 -12637.559,E2 -12637.559} C_VEL
LIN {X 0,Y 369.31,Z 338.591,A -85,B 0,C 180,E1 -12640.43,E2 -12640.43} C_VEL
LIN {X 0,Y 369.701,Z 341.519,A -85,B 0,C 180,E1 -12643.749,E2 -12643.749} C_VEL
LIN {X 0,Y 369.972,Z 344.487,A -85,B 0,C 180,E1 -12646.854,E2 -12646.854} C_VEL
LIN {X 0,Y 369.816,Z 347.5,A -85,B 0,C 180,E1 -12649.749,E2 -12649.749} C_VEL
LIN {X 0,Y 369.513,Z 351.141,A -85,B 0,C 180,E1 -12653.019,E2 -12653.019} C_VEL
LIN {X 0,Y 369.054,Z 355.237,A -85,B 0,C 180,E1 -12656.478,E2 -12656.478} C_VEL
LIN {X 0,Y 368.754,Z 358.424,A -85,B 0,C 180,E1 -12659.054,E2 -12659.054} C_VEL
LIN {X 0,Y 368.295,Z 363.168,A -85,B 0,C 180,E1 -12662.743,E2 -12662.743} C_VEL
LIN {X 0,Y 367.959,Z 368.151,A -85,B 0,C 180,E1 -12666.464,E2 -12666.464} C_VEL
LIN {X 0,Y 367.658,Z 373.51,A -85,B 0,C 180,E1 -12670.348,E2 -12670.348} C_VEL
LIN {X 0,Y 369.811,Z 383.807,A -85,B 0,C 180,E1 -12670.823,E2 -12670.823} C_VEL
LIN {X 0,Y 371.532,Z 393.17,A -85,B 0,C 180,E1 -12671.368,E2 -12671.368} C_VEL
LIN {X 0,Y 372.845,Z 402.504,A -85,B 0,C 180,E1 -12672.014,E2 -12672.014} C_VEL
LIN {X 0,Y 373.408,Z 408.512,A -85,B 0,C 180,E1 -12672.474,E2 -12672.474} C_VEL
LIN {X 0,Y 372.514,Z 419.425,A -85,B 0,C 180,E1 -12673.42,E2 -12673.42} C_VEL
LIN {X 0,Y 371.598,Z 428.37,A -85,B 0,C 180,E1 -12674.365,E2 -12674.365} C_VEL
LIN {X 0,Y 370.905,Z 435.609,A -85,B 0,C 180,E1 -12675.271,E2 -12675.271} C_VEL
LIN {X 0,Y 370.133,Z 444.125,A -85,B 0,C 180,E1 -12676.55,E2 -12676.55} C_VEL
LIN {X 0,Y 369.441,Z 450.326,A -85,B 0,C 180,E1 -12677.642,E2 -12677.642} C_VEL
LIN {X 0,Y 368.725,Z 456.863,A -85,B 0,C 180,E1 -12679.012,E2 -12679.012} C_VEL
LIN {X 0,Y 368.314,Z 461.366,A -85,B 0,C 180,E1 -12680.111,E2 -12680.111} C_VEL
LIN {X 0,Y 367.877,Z 466.859,A -85,B 0,C 180,E1 -12681.762,E2 -12681.762} C_VEL
LIN {X 0,Y 367.566,Z 471.183,A -85,B 0,C 180,E1 -12683.412,E2 -12683.412} C_VEL
LIN {X 0,Y 367.47,Z 473.551,A -85,B 0,C 180,E1 -12684.513,E2 -12684.513} C_VEL
LIN {X 0,Y 367.459,Z 475.351,A -85,B 0,C 180,E1 -12685.612,E2 -12685.612} C_VEL
LIN {X 0,Y 367.36,Z 477.795,A -85,B 0,C 180,E1 -12687.807,E2 -12687.807} C_VEL
LIN {X 0,Y 367.403,Z 478.385,A -85,B 0,C 180,E1 -12688.904,E2 -12688.904} C_VEL
LIN {X 0,Y 367.403,Z 478.385,A -85,B 0,C 180,E1 -12691.096,E2 -12691.096} C_VEL
LIN {X 0,Y 367.36,Z 477.795,A -85,B 0,C 180,E1 -12692.193,E2 -12692.193} C_VEL
LIN {X 0,Y 367.458,Z 475.351,A -85,B 0,C 180,E1 -12694.388,E2 -12694.388} C_VEL
LIN {X 0,Y 367.481,Z 472.452,A -85,B 0,C 180,E1 -12696.014,E2 -12696.014} C_VEL
LIN {X 0,Y 367.735,Z 468.412,A -85,B 0,C 180,E1 -12697.688,E2 -12697.688} C_VEL
LIN {X 0,Y 368.16,Z 463.283,A -85,B 0,C 180,E1 -12699.338,E2 -12699.338} C_VEL
LIN {X 0,Y 368.624,Z 458.019,A -85,B 0,C 180,E1 -12700.713,E2 -12700.713} C_VEL
LIN {X 0,Y 369.265,Z 451.702,A -85,B 0,C 180,E1 -12702.085,E2 -12702.085} C_VEL
LIN {X 0,Y 369.939,Z 445.751,A -85,B 0,C 180,E1 -12703.178,E2 -12703.178} C_VEL
LIN {X 0,Y 370.575,Z 438.821,A -85,B 0,C 180,E1 -12704.273,E2 -12704.273} C_VEL
LIN {X 0,Y 371.335,Z 430.638,A -85,B 0,C 180,E1 -12705.365,E2 -12705.365} C_VEL
LIN {X 0,Y 372.203,Z 422.128,A -85,B 0,C 180,E1 -12706.312,E2 -12706.312} C_VEL
LIN {X 0,Y 373.039,Z 413.412,A -85,B 0,C 180,E1 -12707.12,E2 -12707.12} C_VEL
LIN {X 0,Y 373.385,Z 407.426,A -85,B 0,C 180,E1 -12707.614,E2 -12707.614} C_VEL
LIN {X 0,Y 371.914,Z 395.42,A -85,B 0,C 180,E1 -12708.489,E2 -12708.489} C_VEL
LIN {X 0,Y 370.036,Z 384.731,A -85,B 0,C 180,E1 -12709.127,E2 -12709.127} C_VEL
LIN {X 0,Y 367.683,Z 373.424,A -85,B 0,C 180,E1 -12709.684,E2 -12709.684} C_VEL
LIN {X 0,Y 367.962,Z 367.992,A -85,B 0,C 180,E1 -12713.647,E2 -12713.647} C_VEL
LIN {X 0,Y 368.314,Z 363.164,A -85,B 0,C 180,E1 -12717.255,E2 -12717.255} C_VEL
LIN {X 0,Y 368.757,Z 358.381,A -85,B 0,C 180,E1 -12720.969,E2 -12720.969} C_VEL
LIN {X 0,Y 369.211,Z 353.667,A -85,B 0,C 180,E1 -12724.824,E2 -12724.824} C_VEL
LIN {X 0,Y 369.528,Z 350.564,A -85,B 0,C 180,E1 -12727.488,E2 -12727.488} C_VEL
LIN {X 0,Y 369.849,Z 347.197,A -85,B 0,C 180,E1 -12730.527,E2 -12730.527} C_VEL
LIN {X 0,Y 369.971,Z 344.47,A -85,B 0,C 180,E1 -12733.146,E2 -12733.146} C_VEL
LIN {X 0,Y 369.697,Z 341.519,A -85,B 0,C 180,E1 -12736.251,E2 -12736.251} C_VEL
LIN {X 0,Y 369.277,Z 338.503,A -85,B 0,C 180,E1 -12739.678,E2 -12739.678} C_VEL
LIN {X 0,Y 368.946,Z 336.299,A -85,B 0,C 180,E1 -12742.441,E2 -12742.441} C_VEL
LIN {X 0,Y 368.937,Z 336.032,A -85,B 0,C 180,E1 -12745.146,E2 -12745.146} C_VEL
LIN {X 0,Y 368.93,Z 336.026,A -85,B 0,C 180,E1 -12749.046,E2 -12749.046} C_VEL
LIN {X 0,Y 368.969,Z 336.021,A -85,B 0,C 180,E1 -12752.796,E2 -12752.796} C_VEL
LIN {X 0,Y 368.934,Z 336.028,A -85,B 0,C 180,E1 -12756.116,E2 -12756.116} C_VEL
LIN {X 0,Y 368.938,Z 336.028,A -85,B 0,C 180,E1 -12759.947,E2 -12759.947} C_VEL
LIN {X 0,Y 368.969,Z 336.026,A -85,B 0,C 180,E1 -12763.398,E2 -12763.398} C_VEL
LIN {X 0,Y 369.058,Z 336.011,A -85,B 0,C 180,E1 -12766.79,E2 -12766.79} C_VEL
LIN {X 0,Y 369.067,Z 336.009,A -85,B 0,C 180,E1 -12770.131,E2 -12770.131} C_VEL
LIN {X 0,Y 369.161,Z 335.997,A -85,B 0,C 180,E1 -12772.341,E2 -12772.341} C_VEL
LIN {X 0,Y 369.141,Z 336,A -85,B 0,C 180,E1 -12774.537,E2 -12774.537} C_VEL
LIN {X 0,Y 369.318,Z 335.979,A -85,B 0,C 180,E1 -12777.818,E2 -12777.818} C_VEL
LIN {X 0,Y 369.456,Z 335.961,A -85,B 0,C 180,E1 -12779.999,E2 -12779.999} C_VEL
LIN {X 0,Y 369.318,Z 335.978,A -85,B 0,C 180,E1 -12782.181,E2 -12782.181} C_VEL
LIN {X 0,Y 369.197,Z 335.995,A -85,B 0,C 180,E1 -12786.558,E2 -12786.558} C_VEL
LIN {X 0,Y 369.12,Z 336.006,A -85,B 0,C 180,E1 -12788.761,E2 -12788.761} C_VEL
LIN {X 0,Y 369.003,Z 336.017,A -85,B 0,C 180,E1 -12792.093,E2 -12792.093} C_VEL
LIN {X 0,Y 368.996,Z 336.018,A -85,B 0,C 180,E1 -12795.464,E2 -12795.464} C_VEL
LIN {X 0,Y 368.98,Z 336.024,A -85,B 0,C 180,E1 -12798.892,E2 -12798.892} C_VEL
LIN {X 0,Y 368.923,Z 336.031,A -85,B 0,C 180,E1 -12802.395,E2 -12802.395} C_VEL
LIN {X 0,Y 368.997,Z 336.019,A -85,B 0,C 180,E1 -12805.98,E2 -12805.98} C_VEL
LIN {X 0,Y 368.958,Z 336.025,A -85,B 0,C 180,E1 -12808.811,E2 -12808.811} C_VEL
LIN {X 0,Y 368.899,Z 336.034,A -85,B 0,C 180,E1 -12812.237,E2 -12812.237} C_VEL
LIN {X 0,Y 368.926,Z 336.027,A -85,B 0,C 180,E1 -12815.001,E2 -12815.001} C_VEL
LIN {X 0,Y 368.909,Z 336.031,A -85,B 0,C 180,E1 -12818.641,E2 -12818.641} C_VEL
LIN {X 0,Y 368.948,Z 336.029,A -85,B 0,C 180,E1 -12822.021,E2 -12822.021} C_VEL
LIN {X 0,Y 368.921,Z 336.027,A -85,B 0,C 180,E1 -12825.182,E2 -12825.182} C_VEL
LIN {X 0,Y 368.907,Z 336.033,A -85,B 0,C 180,E1 -12828.181,E2 -12828.181} C_VEL
LIN {X 0,Y 368.909,Z 336.03,A -85,B 0,C 180,E1 -12831.359,E2 -12831.359} C_VEL
LIN {X 0,Y 368.933,Z 336.026,A -85,B 0,C 180,E1 -12835.146,E2 -12835.146} C_VEL
LIN {X 0,Y 368.925,Z 336.027,A -85,B 0,C 180,E1 -12839.046,E2 -12839.046} C_VEL
LIN {X 0,Y 368.976,Z 336.025,A -85,B 0,C 180,E1 -12841.564,E2 -12841.564} C_VEL
LIN {X 0,Y 368.996,Z 336.02,A -85,B 0,C 180,E1 -12844.02,E2 -12844.02} C_VEL
LIN {X 0,Y 368.93,Z 336.032,A -85,B 0,C 180,E1 -12847.605,E2 -12847.605} C_VEL
LIN {X 0,Y 368.98,Z 336.025,A -85,B 0,C 180,E1 -12851.107,E2 -12851.107} C_VEL
LIN {X 0,Y 369.003,Z 336.022,A -85,B 0,C 180,E1 -12855.101,E2 -12855.101} C_VEL
LIN {X 0,Y 369.007,Z 336.064,A -85,B 0,C 180,E1 -12855.418,E2 -12855.418} C_VEL
LIN {X 0,Y 369.856,Z 338.615,A -85,B 0,C 180,E1 -12855.717,E2 -12855.717} C_VEL
LIN {X 0,Y 371.771,Z 340.779,A -85,B 0,C 180,E1 -12856.311,E2 -12856.311} C_VEL
LIN {X 0,Y 373.673,Z 341.974,A -85,B 0,C 180,E1 -12856.887,E2 -12856.887} C_VEL
LIN {X 0,Y 375.511,Z 345.026,A -85,B 0,C 180,E1 -12857.536,E2 -12857.536} C_VEL
LIN {X 0,Y 378.018,Z 347.219,A -85,B 0,C 180,E1 -12858.419,E2 -12858.419} C_VEL
LIN {X 0,Y 379.35,Z 348.061,A -85,B 0,C 180,E1 -12858.896,E2 -12858.896} C_VEL
LIN {X 0,Y 381.255,Z 350.949,A -85,B 0,C 180,E1 -12859.713,E2 -12859.713} C_VEL
LIN {X 0,Y 384.014,Z 353.228,A -85,B 0,C 180,E1 -12860.918,E2 -12860.918} C_VEL
LIN {X 0,Y 386.046,Z 354.315,A -85,B 0,C 180,E1 -12861.883,E2 -12861.883} C_VEL
LIN {X 0,Y 387.951,Z 357.16,A -85,B 0,C 180,E1 -12863.039,E2 -12863.039} C_VEL
LIN {X 0,Y 389.99,Z 359.136,A -85,B 0,C 180,E1 -12864.441,E2 -12864.441} C_VEL
LIN {X 0,Y 391.644,Z 360.134,A -85,B 0,C 180,E1 -12865.884,E2 -12865.884} C_VEL
LIN {X 0,Y 393.22,Z 360.524,A -85,B 0,C 180,E1 -12867.951,E2 -12867.951} C_VEL
LIN {X 0,Y 393.637,Z 360.553,A -85,B 0,C 180,E1 -12868.977,E2 -12868.977} C_VEL
LIN {X 0,Y 393.779,Z 360.579,A -85,B 0,C 180,E1 -12870,E2 -12870} C_VEL
LIN {X 0,Y 393.63,Z 360.554,A -85,B 0,C 180,E1 -12871.061,E2 -12871.061} C_VEL
LIN {X 0,Y 392.568,Z 360.346,A -85,B 0,C 180,E1 -12873.079,E2 -12873.079} C_VEL
LIN {X 0,Y 391.09,Z 359.881,A -85,B 0,C 180,E1 -12874.638,E2 -12874.638} C_VEL
LIN {X 0,Y 389.048,Z 358.377,A -85,B 0,C 180,E1 -12876.222,E2 -12876.222} C_VEL
LIN {X 0,Y 386.851,Z 355.733,A -85,B 0,C 180,E1 -12877.627,E2 -12877.627} C_VEL
LIN {X 0,Y 385.902,Z 354.062,A -85,B 0,C 180,E1 -12878.206,E2 -12878.206} C_VEL
LIN {X 0,Y 383.077,Z 352.61,A -85,B 0,C 180,E1 -12879.504,E2 -12879.504} C_VEL
LIN {X 0,Y 380.566,Z 350.106,A -85,B 0,C 180,E1 -12880.575,E2 -12880.575} C_VEL
LIN {X 0,Y 379.094,Z 347.76,A -85,B 0,C 180,E1 -12881.204,E2 -12881.204} C_VEL
LIN {X 0,Y 376.337,Z 345.955,A -85,B 0,C 180,E1 -12882.162,E2 -12882.162} C_VEL
LIN {X 0,Y 374.313,Z 343.266,A -85,B 0,C 180,E1 -12882.888,E2 -12882.888} C_VEL
LIN {X 0,Y 373.605,Z 341.795,A -85,B 0,C 180,E1 -12883.139,E2 -12883.139} C_VEL
LIN {X 0,Y 370.881,Z 339.987,A -85,B 0,C 180,E1 -12883.966,E2 -12883.966} C_VEL
LIN {X 0,Y 369.476,Z 337.814,A -85,B 0,C 180,E1 -12884.404,E2 -12884.404} C_VEL
LIN {X 0,Y 369.016,Z 336.022,A -85,B 0,C 180,E1 -12884.617,E2 -12884.617} C_VEL
LIN {X 0,Y 368.997,Z 336.022,A -85,B 0,C 180,E1 -12887.768,E2 -12887.768} C_VEL
LIN {X 0,Y 368.926,Z 336.027,A -85,B 0,C 180,E1 -12891.22,E2 -12891.22} C_VEL
LIN {X 0,Y 368.954,Z 336.026,A -85,B 0,C 180,E1 -12894.775,E2 -12894.775} C_VEL
LIN {X 0,Y 368.964,Z 336.022,A -85,B 0,C 180,E1 -12897.203,E2 -12897.203} C_VEL
LIN {X 0,Y 368.915,Z 336.029,A -85,B 0,C 180,E1 -12899.69,E2 -12899.69} C_VEL
LIN {X 0,Y 368.895,Z 336.03,A -85,B 0,C 180,E1 -12903.044,E2 -12903.044} C_VEL
LIN {X 0,Y 368.915,Z 336.034,A -85,B 0,C 180,E1 -12906.197,E2 -12906.197} C_VEL
LIN {X 0,Y 368.918,Z 336.027,A -85,B 0,C 180,E1 -12910.031,E2 -12910.031} C_VEL
LIN {X 0,Y 368.897,Z 336.033,A -85,B 0,C 180,E1 -12913.619,E2 -12913.619} C_VEL
LIN {X 0,Y 368.916,Z 336.027,A -85,B 0,C 180,E1 -12914.755,E2 -12914.755} C_VEL
LIN {X 0,Y 368.309,Z 336.108,A -85,B 0,C 180,E1 -12915.666,E2 -12915.666} C_VEL
LIN {X 0,Y 365.481,Z 336.46,A -85,B 0,C 180,E1 -12917.148,E2 -12917.148} C_VEL
LIN {X 0,Y 363.04,Z 336.761,A -85,B 0,C 180,E1 -12918.346,E2 -12918.346} C_VEL
LIN {X 0,Y 361.975,Z 336.894,A -85,B 0,C 180,E1 -12919.273,E2 -12919.273} C_VEL
LIN {X 0,Y 361.882,Z 336.904,A -85,B 0,C 180,E1 -12919.587,E2 -12919.587} C_VEL
LIN {X 0,Y 361.866,Z 336.906,A -85,B 0,C 180,E1 -12922.983,E2 -12922.983} C_VEL
LIN {X 0,Y 361.858,Z 336.907,A -85,B 0,C 180,E1 -12926.631,E2 -12926.631} C_VEL
LIN {X 0,Y 361.872,Z 336.91,A -85,B 0,C 180,E1 -12929.673,E2 -12929.673} C_VEL
LIN {X 0,Y 361.952,Z 336.902,A -85,B 0,C 180,E1 -12933.476,E2 -12933.476} C_VEL
LIN {X 0,Y 361.88,Z 336.908,A -85,B 0,C 180,E1 -12937.145,E2 -12937.145} C_VEL
LIN {X 0,Y 361.919,Z 336.901,A -85,B 0,C 180,E1 -12940.725,E2 -12940.725} C_VEL
LIN {X 0,Y 361.944,Z 336.896,A -85,B 0,C 180,E1 -12944.227,E2 -12944.227} C_VEL
LIN {X 0,Y 361.997,Z 336.891,A -85,B 0,C 180,E1 -12946.528,E2 -12946.528} C_VEL
LIN {X 0,Y 362.03,Z 336.886,A -85,B 0,C 180,E1 -12949.939,E2 -12949.939} C_VEL
LIN {X 0,Y 362.159,Z 336.872,A -85,B 0,C 180,E1 -12953.314,E2 -12953.314} C_VEL
LIN {X 0,Y 362.282,Z 336.854,A -85,B 0,C 180,E1 -12957.777,E2 -12957.777} C_VEL
LIN {X 0,Y 362.425,Z 336.836,A -85,B 0,C 180,E1 -12960.001,E2 -12960.001} C_VEL
LIN {X 0,Y 362.282,Z 336.855,A -85,B 0,C 180,E1 -12962.224,E2 -12962.224} C_VEL
LIN {X 0,Y 362.16,Z 336.875,A -85,B 0,C 180,E1 -12966.687,E2 -12966.687} C_VEL
LIN {X 0,Y 362.031,Z 336.887,A -85,B 0,C 180,E1 -12970.063,E2 -12970.063} C_VEL
LIN {X 0,Y 361.998,Z 336.891,A -85,B 0,C 180,E1 -12973.899,E2 -12973.899} C_VEL
LIN {X 0,Y 361.928,Z 336.9,A -85,B 0,C 180,E1 -12976.935,E2 -12976.935} C_VEL
LIN {X 0,Y 361.888,Z 336.908,A -85,B 0,C 180,E1 -12980.461,E2 -12980.461} C_VEL
LIN {X 0,Y 361.893,Z 336.908,A -85,B 0,C 180,E1 -12984.113,E2 -12984.113} C_VEL
LIN {X 0,Y 361.943,Z 336.898,A -85,B 0,C 180,E1 -12986.722,E2 -12986.722} C_VEL
LIN {X 0,Y 361.874,Z 336.909,A -85,B 0,C 180,E1 -12990.329,E2 -12990.329} C_VEL
LIN {X 0,Y 361.855,Z 336.914,A -85,B 0,C 180,E1 -12994.281,E2 -12994.281} C_VEL
LIN {X 0,Y 361.906,Z 337.187,A -85,B 0,C 180,E1 -12997.232,E2 -12997.232} C_VEL
LIN {X 0,Y 362.397,Z 340.41,A -85,B 0,C 180,E1 -13001.252,E2 -13001.252} C_VEL
LIN {X 0,Y 362.737,Z 342.99,A -85,B 0,C 180,E1 -13004.227,E2 -13004.227} C_VEL
LIN {X 0,Y 362.918,Z 346.005,A -85,B 0,C 180,E1 -13007.382,E2 -13007.382} C_VEL
LIN {X 0,Y 362.695,Z 349.576,A -85,B 0,C 180,E1 -13010.814,E2 -13010.814} C_VEL
LIN {X 0,Y 362.451,Z 352.052,A -85,B 0,C 180,E1 -13013.052,E2 -13013.052} C_VEL
LIN {X 0,Y 361.917,Z 356.723,A -85,B 0,C 180,E1 -13017.063,E2 -13017.063} C_VEL
LIN {X 0,Y 361.44,Z 361.467,A -85,B 0,C 180,E1 -13020.915,E2 -13020.915} C_VEL
LIN {X 0,Y 361.02,Z 366.249,A -85,B 0,C 180,E1 -13024.642,E2 -13024.642} C_VEL
LIN {X 0,Y 360.698,Z 371.076,A -85,B 0,C 180,E1 -13028.272,E2 -13028.272} C_VEL
LIN {X 0,Y 360.59,Z 373.303,A -85,B 0,C 180,E1 -13029.946,E2 -13029.946} C_VEL
LIN {X 0,Y 362.833,Z 383.889,A -85,B 0,C 180,E1 -13030.452,E2 -13030.452} C_VEL
LIN {X 0,Y 364.734,Z 394.106,A -85,B 0,C 180,E1 -13031.071,E2 -13031.071} C_VEL
LIN {X 0,Y 366.236,Z 405.084,A -85,B 0,C 180,E1 -13031.876,E2 -13031.876} C_VEL
LIN {X 0,Y 366.501,Z 409.95,A -85,B 0,C 180,E1 -13032.277,E2 -13032.277} C_VEL
LIN {X 0,Y 365.669,Z 419.228,A -85,B 0,C 180,E1 -13033.1,E2 -13033.1} C_VEL
LIN {X 0,Y 364.738,Z 428.173,A -85,B 0,C 180,E1 -13034.063,E2 -13034.063} C_VEL
LIN {X 0,Y 363.927,Z 436.195,A -85,B 0,C 180,E1 -13035.098,E2 -13035.098} C_VEL
LIN {X 0,Y 363.201,Z 443.928,A -85,B 0,C 180,E1 -13036.288,E2 -13036.288} C_VEL
LIN {X 0,Y 362.473,Z 450.13,A -85,B 0,C 180,E1 -13037.401,E2 -13037.401} C_VEL
LIN {X 0,Y 361.712,Z 456.666,A -85,B 0,C 180,E1 -13038.796,E2 -13038.796} C_VEL
LIN {X 0,Y 361.278,Z 461.169,A -85,B 0,C 180,E1 -13039.917,E2 -13039.917} C_VEL
LIN {X 0,Y 360.823,Z 466.662,A -85,B 0,C 180,E1 -13041.6,E2 -13041.6} C_VEL
LIN {X 0,Y 360.501,Z 470.987,A -85,B 0,C 180,E1 -13043.283,E2 -13043.283} C_VEL
LIN {X 0,Y 360.39,Z 473.355,A -85,B 0,C 180,E1 -13044.404,E2 -13044.404} C_VEL
LIN {X 0,Y 360.368,Z 475.155,A -85,B 0,C 180,E1 -13045.526,E2 -13045.526} C_VEL
LIN {X 0,Y 360.265,Z 477.599,A -85,B 0,C 180,E1 -13047.764,E2 -13047.764} C_VEL
LIN {X 0,Y 360.303,Z 478.189,A -85,B 0,C 180,E1 -13048.882,E2 -13048.882} C_VEL
LIN {X 0,Y 360.303,Z 478.189,A -85,B 0,C 180,E1 -13051.118,E2 -13051.118} C_VEL
LIN {X 0,Y 360.265,Z 477.599,A -85,B 0,C 180,E1 -13052.236,E2 -13052.236} C_VEL
LIN {X 0,Y 360.367,Z 475.155,A -85,B 0,C 180,E1 -13054.474,E2 -13054.474} C_VEL
LIN {X 0,Y 360.38,Z 472.629,A -85,B 0,C 180,E1 -13055.961,E2 -13055.961} C_VEL
LIN {X 0,Y 360.597,Z 469.747,A -85,B 0,C 180,E1 -13057.278,E2 -13057.278} C_VEL
LIN {X 0,Y 360.96,Z 465.002,A -85,B 0,C 180,E1 -13058.961,E2 -13058.961} C_VEL
LIN {X 0,Y 361.518,Z 458.979,A -85,B 0,C 180,E1 -13060.643,E2 -13060.643} C_VEL
LIN {X 0,Y 362.123,Z 452.881,A -85,B 0,C 180,E1 -13062.042,E2 -13062.042} C_VEL
LIN {X 0,Y 362.818,Z 447.182,A -85,B 0,C 180,E1 -13063.156,E2 -13063.156} C_VEL
LIN {X 0,Y 363.682,Z 438.625,A -85,B 0,C 180,E1 -13064.55,E2 -13064.55} C_VEL
LIN {X 0,Y 364.469,Z 430.442,A -85,B 0,C 180,E1 -13065.662,E2 -13065.662} C_VEL
LIN {X 0,Y 365.388,Z 421.931,A -85,B 0,C 180,E1 -13066.625,E2 -13066.625} C_VEL
LIN {X 0,Y 366.233,Z 413.215,A -85,B 0,C 180,E1 -13067.448,E2 -13067.448} C_VEL
LIN {X 0,Y 366.423,Z 407.318,A -85,B 0,C 180,E1 -13067.953,E2 -13067.953} C_VEL
LIN {X 0,Y 364.982,Z 395.721,A -85,B 0,C 180,E1 -13068.825,E2 -13068.825} C_VEL
LIN {X 0,Y 362.99,Z 384.407,A -85,B 0,C 180,E1 -13069.518,E2 -13069.518} C_VEL
LIN {X 0,Y 360.678,Z 373.805,A -85,B 0,C 180,E1 -13070.035,E2 -13070.035} C_VEL
LIN {X 0,Y 360.632,Z 373.252,A -85,B 0,C 180,E1 -13070.089,E2 -13070.089} C_VEL
LIN {X 0,Y 360.914,Z 367.848,A -85,B 0,C 180,E1 -13074.137,E2 -13074.137} C_VEL
LIN {X 0,Y 361.299,Z 363.038,A -85,B 0,C 180,E1 -13077.83,E2 -13077.83} C_VEL
LIN {X 0,Y 361.735,Z 358.284,A -85,B 0,C 180,E1 -13081.639,E2 -13081.639} C_VEL
LIN {X 0,Y 362.075,Z 355.152,A -85,B 0,C 180,E1 -13084.256,E2 -13084.256} C_VEL
LIN {X 0,Y 362.472,Z 351.594,A -85,B 0,C 180,E1 -13087.348,E2 -13087.348} C_VEL
LIN {X 0,Y 362.707,Z 348.976,A -85,B 0,C 180,E1 -13089.749,E2 -13089.749} C_VEL
LIN {X 0,Y 362.946,Z 345.94,A -85,B 0,C 180,E1 -13092.666,E2 -13092.666} C_VEL
LIN {X 0,Y 362.733,Z 342.965,A -85,B 0,C 180,E1 -13095.797,E2 -13095.797} C_VEL
LIN {X 0,Y 362.344,Z 340.069,A -85,B 0,C 180,E1 -13099.151,E2 -13099.151} C_VEL
LIN {X 0,Y 361.88,Z 337.031,A -85,B 0,C 180,E1 -13102.983,E2 -13102.983} C_VEL
LIN {X 0,Y 361.86,Z 336.908,A -85,B 0,C 180,E1 -13106.63,E2 -13106.63} C_VEL
LIN {X 0,Y 361.874,Z 336.909,A -85,B 0,C 180,E1 -13109.671,E2 -13109.671} C_VEL
LIN {X 0,Y 361.955,Z 336.898,A -85,B 0,C 180,E1 -13113.475,E2 -13113.475} C_VEL
LIN {X 0,Y 361.88,Z 336.905,A -85,B 0,C 180,E1 -13117.143,E2 -13117.143} C_VEL
LIN {X 0,Y 361.887,Z 336.903,A -85,B 0,C 180,E1 -13120.722,E2 -13120.722} C_VEL
LIN {X 0,Y 361.944,Z 336.897,A -85,B 0,C 180,E1 -13124.225,E2 -13124.225} C_VEL
LIN {X 0,Y 361.999,Z 336.889,A -85,B 0,C 180,E1 -13126.527,E2 -13126.527} C_VEL
LIN {X 0,Y 362.031,Z 336.887,A -85,B 0,C 180,E1 -13129.937,E2 -13129.937} C_VEL
LIN {X 0,Y 362.16,Z 336.875,A -85,B 0,C 180,E1 -13133.313,E2 -13133.313} C_VEL
LIN {X 0,Y 362.281,Z 336.855,A -85,B 0,C 180,E1 -13137.776,E2 -13137.776} C_VEL
LIN {X 0,Y 362.425,Z 336.836,A -85,B 0,C 180,E1 -13139.999,E2 -13139.999} C_VEL
LIN {X 0,Y 362.282,Z 336.854,A -85,B 0,C 180,E1 -13142.223,E2 -13142.223} C_VEL
LIN {X 0,Y 362.159,Z 336.872,A -85,B 0,C 180,E1 -13146.686,E2 -13146.686} C_VEL
LIN {X 0,Y 362.03,Z 336.886,A -85,B 0,C 180,E1 -13150.061,E2 -13150.061} C_VEL
LIN {X 0,Y 361.996,Z 336.89,A -85,B 0,C 180,E1 -13153.898,E2 -13153.898} C_VEL
LIN {X 0,Y 361.965,Z 336.894,A -85,B 0,C 180,E1 -13157.938,E2 -13157.938} C_VEL
LIN {X 0,Y 361.859,Z 336.907,A -85,B 0,C 180,E1 -13161.654,E2 -13161.654} C_VEL
LIN {X 0,Y 361.924,Z 336.899,A -85,B 0,C 180,E1 -13165.29,E2 -13165.29} C_VEL
LIN {X 0,Y 361.915,Z 336.9,A -85,B 0,C 180,E1 -13167.778,E2 -13167.778} C_VEL
LIN {X 0,Y 361.844,Z 336.909,A -85,B 0,C 180,E1 -13171.285,E2 -13171.285} C_VEL
LIN {X 0,Y 361.853,Z 336.913,A -85,B 0,C 180,E1 -13174.28,E2 -13174.28} C_VEL
LIN {X 0,Y 361.862,Z 336.906,A -85,B 0,C 180,E1 -13177.223,E2 -13177.223} C_VEL
LIN {X 0,Y 361.903,Z 336.902,A -85,B 0,C 180,E1 -13180.768,E2 -13180.768} C_VEL
LIN {X 0,Y 361.908,Z 336.904,A -85,B 0,C 180,E1 -13184.353,E2 -13184.353} C_VEL
LIN {X 0,Y 361.854,Z 336.909,A -85,B 0,C 180,E1 -13187.564,E2 -13187.564} C_VEL
LIN {X 0,Y 361.871,Z 336.905,A -85,B 0,C 180,E1 -13190.972,E2 -13190.972} C_VEL
LIN {X 0,Y 361.871,Z 336.906,A -85,B 0,C 180,E1 -13194.655,E2 -13194.655} C_VEL
LIN {X 0,Y 361.834,Z 336.911,A -85,B 0,C 180,E1 -13198.37,E2 -13198.37} C_VEL
LIN {X 0,Y 361.896,Z 336.903,A -85,B 0,C 180,E1 -13200.955,E2 -13200.955} C_VEL
LIN {X 0,Y 361.951,Z 336.9,A -85,B 0,C 180,E1 -13203.475,E2 -13203.475} C_VEL
LIN {X 0,Y 361.887,Z 336.906,A -85,B 0,C 180,E1 -13207.145,E2 -13207.145} C_VEL
LIN {X 0,Y 361.918,Z 336.904,A -85,B 0,C 180,E1 -13210.724,E2 -13210.724} C_VEL
LIN {X 0,Y 361.932,Z 336.902,A -85,B 0,C 180,E1 -13213.755,E2 -13213.755} C_VEL
LIN {X 0,Y 362.913,Z 339.73,A -85,B 0,C 180,E1 -13214.095,E2 -13214.095} C_VEL
LIN {X 0,Y 364.909,Z 341.824,A -85,B 0,C 180,E1 -13214.617,E2 -13214.617} C_VEL
LIN {X 0,Y 366.277,Z 342.771,A -85,B 0,C 180,E1 -13214.978,E2 -13214.978} C_VEL
LIN {X 0,Y 368.036,Z 345.697,A -85,B 0,C 180,E1 -13215.52,E2 -13215.52} C_VEL
LIN {X 0,Y 370.628,Z 347.898,A -85,B 0,C 180,E1 -13216.268,E2 -13216.268} C_VEL
LIN {X 0,Y 371.686,Z 348.942,A -85,B 0,C 180,E1 -13216.605,E2 -13216.605} C_VEL
LIN {X 0,Y 374.012,Z 352.035,A -85,B 0,C 180,E1 -13217.38,E2 -13217.38} C_VEL
LIN {X 0,Y 376.773,Z 354.176,A -85,B 0,C 180,E1 -13218.325,E2 -13218.325} C_VEL
LIN {X 0,Y 377.724,Z 355.085,A -85,B 0,C 180,E1 -13218.664,E2 -13218.664} C_VEL
LIN {X 0,Y 380.045,Z 358.027,A -85,B 0,C 180,E1 -13219.613,E2 -13219.613} C_VEL
LIN {X 0,Y 382.715,Z 360.114,A -85,B 0,C 180,E1 -13220.746,E2 -13220.746} C_VEL
LIN {X 0,Y 384.738,Z 361.318,A -85,B 0,C 180,E1 -13221.683,E2 -13221.683} C_VEL
LIN {X 0,Y 386.981,Z 364.32,A -85,B 0,C 180,E1 -13223.007,E2 -13223.007} C_VEL
LIN {X 0,Y 388.899,Z 366.054,A -85,B 0,C 180,E1 -13224.296,E2 -13224.296} C_VEL
LIN {X 0,Y 390.755,Z 367.177,A -85,B 0,C 180,E1 -13225.874,E2 -13225.874} C_VEL
LIN {X 0,Y 392.358,Z 367.566,A -85,B 0,C 180,E1 -13227.947,E2 -13227.947} C_VEL
LIN {X 0,Y 392.776,Z 367.6,A -85,B 0,C 180,E1 -13228.975,E2 -13228.975} C_VEL
LIN {X 0,Y 392.914,Z 367.626,A -85,B 0,C 180,E1 -13230,E2 -13230} C_VEL
LIN {X 0,Y 392.776,Z 367.603,A -85,B 0,C 180,E1 -13231.025,E2 -13231.025} C_VEL
LIN {X 0,Y 391.691,Z 367.391,A -85,B 0,C 180,E1 -13233.086,E2 -13233.086} C_VEL
LIN {X 0,Y 390.205,Z 366.907,A -85,B 0,C 180,E1 -13234.649,E2 -13234.649} C_VEL
LIN {X 0,Y 387.984,Z 365.371,A -85,B 0,C 180,E1 -13236.337,E2 -13236.337} C_VEL
LIN {X 0,Y 385.689,Z 362.763,A -85,B 0,C 180,E1 -13237.758,E2 -13237.758} C_VEL
LIN {X 0,Y 384.275,Z 360.856,A -85,B 0,C 180,E1 -13238.546,E2 -13238.546} C_VEL
LIN {X 0,Y 381.278,Z 359.11,A -85,B 0,C 180,E1 -13239.884,E2 -13239.884} C_VEL
LIN {X 0,Y 378.546,Z 356.304,A -85,B 0,C 180,E1 -13241,E2 -13241} C_VEL
LIN {X 0,Y 377.317,Z 354.469,A -85,B 0,C 180,E1 -13241.493,E2 -13241.493} C_VEL
LIN {X 0,Y 374.248,Z 352.255,A -85,B 0,C 180,E1 -13242.541,E2 -13242.541} C_VEL
LIN {X 0,Y 371.834,Z 349.223,A -85,B 0,C 180,E1 -13243.343,E2 -13243.343} C_VEL
LIN {X 0,Y 370.87,Z 348.042,A -85,B 0,C 180,E1 -13243.658,E2 -13243.658} C_VEL
LIN {X 0,Y 368.151,Z 345.832,A -85,B 0,C 180,E1 -13244.447,E2 -13244.447} C_VEL
LIN {X 0,Y 366.335,Z 342.913,A -85,B 0,C 180,E1 -13245.003,E2 -13245.003} C_VEL
LIN {X 0,Y 365.638,Z 342.247,A -85,B 0,C 180,E1 -13245.2,E2 -13245.2} C_VEL
LIN {X 0,Y 363.299,Z 340.281,A -85,B 0,C 180,E1 -13245.8,E2 -13245.8} C_VEL
LIN {X 0,Y 362.124,Z 337.851,A -85,B 0,C 180,E1 -13246.145,E2 -13246.145} C_VEL
LIN {X 0,Y 361.932,Z 336.902,A -85,B 0,C 180,E1 -13246.245,E2 -13246.245} C_VEL
LIN {X 0,Y 361.918,Z 336.904,A -85,B 0,C 180,E1 -13249.276,E2 -13249.276} C_VEL
LIN {X 0,Y 361.887,Z 336.906,A -85,B 0,C 180,E1 -13252.855,E2 -13252.855} C_VEL
LIN {X 0,Y 361.939,Z 336.899,A -85,B 0,C 180,E1 -13256.722,E2 -13256.722} C_VEL
LIN {X 0,Y 361.871,Z 336.911,A -85,B 0,C 180,E1 -13260.328,E2 -13260.328} C_VEL
LIN {X 0,Y 361.851,Z 336.913,A -85,B 0,C 180,E1 -13264.281,E2 -13264.281} C_VEL
LIN {X 0,Y 361.862,Z 336.907,A -85,B 0,C 180,E1 -13267.224,E2 -13267.224} C_VEL
LIN {X 0,Y 361.869,Z 336.906,A -85,B 0,C 180,E1 -13270.763,E2 -13270.763} C_VEL
LIN {X 0,Y 361.862,Z 336.908,A -85,B 0,C 180,E1 -13274.361,E2 -13274.361} C_VEL
LIN {X 0,Y 361.886,Z 336.907,A -85,B 0,C 180,E1 -13277.559,E2 -13277.559} C_VEL
LIN {X 0,Y 361.882,Z 336.904,A -85,B 0,C 180,E1 -13279.587,E2 -13279.587} C_VEL
LIN {X 0,Y 361.199,Z 336.991,A -85,B 0,C 180,E1 -13280.515,E2 -13280.515} C_VEL
LIN {X 0,Y 358.348,Z 337.347,A -85,B 0,C 180,E1 -13282.025,E2 -13282.025} C_VEL
LIN {X 0,Y 355.939,Z 337.647,A -85,B 0,C 180,E1 -13283.247,E2 -13283.247} C_VEL
LIN {X 0,Y 354.899,Z 337.776,A -85,B 0,C 180,E1 -13284.192,E2 -13284.192} C_VEL
LIN {X 0,Y 354.811,Z 337.785,A -85,B 0,C 180,E1 -13284.512,E2 -13284.512} C_VEL
LIN {X 0,Y 354.786,Z 337.794,A -85,B 0,C 180,E1 -13287.667,E2 -13287.667} C_VEL
LIN {X 0,Y 354.866,Z 337.778,A -85,B 0,C 180,E1 -13290.622,E2 -13290.622} C_VEL
LIN {X 0,Y 354.896,Z 337.775,A -85,B 0,C 180,E1 -13294.173,E2 -13294.173} C_VEL
LIN {X 0,Y 354.815,Z 337.786,A -85,B 0,C 180,E1 -13297.893,E2 -13297.893} C_VEL
LIN {X 0,Y 354.921,Z 337.772,A -85,B 0,C 180,E1 -13301.892,E2 -13301.892} C_VEL
LIN {X 0,Y 354.941,Z 337.769,A -85,B 0,C 180,E1 -13305.982,E2 -13305.982} C_VEL
LIN {X 0,Y 354.977,Z 337.765,A -85,B 0,C 180,E1 -13309.737,E2 -13309.737} C_VEL
LIN {X 0,Y 355.124,Z 337.75,A -85,B 0,C 180,E1 -13313.181,E2 -13313.181} C_VEL
LIN {X 0,Y 355.245,Z 337.73,A -85,B 0,C 180,E1 -13317.733,E2 -13317.733} C_VEL
LIN {X 0,Y 355.374,Z 337.715,A -85,B 0,C 180,E1 -13320.001,E2 -13320.001} C_VEL
LIN {X 0,Y 355.245,Z 337.732,A -85,B 0,C 180,E1 -13322.268,E2 -13322.268} C_VEL
LIN {X 0,Y 355.125,Z 337.75,A -85,B 0,C 180,E1 -13326.82,E2 -13326.82} C_VEL
LIN {X 0,Y 354.978,Z 337.767,A -85,B 0,C 180,E1 -13330.265,E2 -13330.265} C_VEL
LIN {X 0,Y 354.943,Z 337.77,A -85,B 0,C 180,E1 -13334.019,E2 -13334.019} C_VEL
LIN {X 0,Y 354.89,Z 337.778,A -85,B 0,C 180,E1 -13338.093,E2 -13338.093} C_VEL
LIN {X 0,Y 354.816,Z 337.789,A -85,B 0,C 180,E1 -13342.108,E2 -13342.108} C_VEL
LIN {X 0,Y 354.899,Z 337.777,A -85,B 0,C 180,E1 -13345.828,E2 -13345.828} C_VEL
LIN {X 0,Y 354.818,Z 337.786,A -85,B 0,C 180,E1 -13349.682,E2 -13349.682} C_VEL
LIN {X 0,Y 354.807,Z 337.789,A -85,B 0,C 180,E1 -13353.703,E2 -13353.703} C_VEL
LIN {X 0,Y 354.801,Z 337.792,A -85,B 0,C 180,E1 -13356.46,E2 -13356.46} C_VEL
LIN {X 0,Y 355.141,Z 340.084,A -85,B 0,C 180,E1 -13359.486,E2 -13359.486} C_VEL
LIN {X 0,Y 355.459,Z 342.308,A -85,B 0,C 180,E1 -13362.24,E2 -13362.24} C_VEL
LIN {X 0,Y 355.805,Z 345.039,A -85,B 0,C 180,E1 -13365.324,E2 -13365.324} C_VEL
LIN {X 0,Y 355.831,Z 348.235,A -85,B 0,C 180,E1 -13368.638,E2 -13368.638} C_VEL
LIN {X 0,Y 355.487,Z 351.978,A -85,B 0,C 180,E1 -13372.203,E2 -13372.203} C_VEL
LIN {X 0,Y 355.102,Z 355.068,A -85,B 0,C 180,E1 -13374.974,E2 -13374.974} C_VEL
LIN {X 0,Y 354.61,Z 359.762,A -85,B 0,C 180,E1 -13378.983,E2 -13378.983} C_VEL
LIN {X 0,Y 354.26,Z 362.928,A -85,B 0,C 180,E1 -13381.568,E2 -13381.568} C_VEL
LIN {X 0,Y 353.858,Z 367.704,A -85,B 0,C 180,E1 -13385.35,E2 -13385.35} C_VEL
LIN {X 0,Y 353.555,Z 373.084,A -85,B 0,C 180,E1 -13389.491,E2 -13389.491} C_VEL
LIN {X 0,Y 353.58,Z 373.613,A -85,B 0,C 180,E1 -13389.546,E2 -13389.546} C_VEL
LIN {X 0,Y 356.002,Z 384.597,A -85,B 0,C 180,E1 -13390.1,E2 -13390.1} C_VEL
LIN {X 0,Y 358.286,Z 397.449,A -85,B 0,C 180,E1 -13390.922,E2 -13390.922} C_VEL
LIN {X 0,Y 359.577,Z 408.111,A -85,B 0,C 180,E1 -13391.777,E2 -13391.777} C_VEL
LIN {X 0,Y 359.319,Z 414.651,A -85,B 0,C 180,E1 -13392.352,E2 -13392.352} C_VEL
LIN {X 0,Y 358.016,Z 426.842,A -85,B 0,C 180,E1 -13393.609,E2 -13393.609} C_VEL
LIN {X 0,Y 357.141,Z 434.855,A -85,B 0,C 180,E1 -13394.635,E2 -13394.635} C_VEL
LIN {X 0,Y 356.266,Z 443.731,A -85,B 0,C 180,E1 -13396.016,E2 -13396.016} C_VEL
LIN {X 0,Y 355.501,Z 449.932,A -85,B 0,C 180,E1 -13397.15,E2 -13397.15} C_VEL
LIN {X 0,Y 354.71,Z 456.469,A -85,B 0,C 180,E1 -13398.572,E2 -13398.572} C_VEL
LIN {X 0,Y 354.265,Z 460.972,A -85,B 0,C 180,E1 -13399.715,E2 -13399.715} C_VEL
LIN {X 0,Y 353.782,Z 466.466,A -85,B 0,C 180,E1 -13401.432,E2 -13401.432} C_VEL
LIN {X 0,Y 353.42,Z 470.791,A -85,B 0,C 180,E1 -13403.148,E2 -13403.148} C_VEL
LIN {X 0,Y 353.312,Z 473.158,A -85,B 0,C 180,E1 -13404.292,E2 -13404.292} C_VEL
LIN {X 0,Y 353.281,Z 474.959,A -85,B 0,C 180,E1 -13405.436,E2 -13405.436} C_VEL
LIN {X 0,Y 353.173,Z 477.403,A -85,B 0,C 180,E1 -13407.719,E2 -13407.719} C_VEL
LIN {X 0,Y 353.204,Z 477.993,A -85,B 0,C 180,E1 -13408.86,E2 -13408.86} C_VEL
LIN {X 0,Y 353.262,Z 478.149,A -85,B 0,C 180,E1 -13410,E2 -13410} C_VEL
LIN {X 0,Y 353.204,Z 477.993,A -85,B 0,C 180,E1 -13411.14,E2 -13411.14} C_VEL
LIN {X 0,Y 353.173,Z 477.403,A -85,B 0,C 180,E1 -13412.281,E2 -13412.281} C_VEL
LIN {X 0,Y 353.28,Z 474.959,A -85,B 0,C 180,E1 -13414.564,E2 -13414.564} C_VEL
LIN {X 0,Y 353.298,Z 472.737,A -85,B 0,C 180,E1 -13415.937,E2 -13415.937} C_VEL
LIN {X 0,Y 353.521,Z 469.55,A -85,B 0,C 180,E1 -13417.424,E2 -13417.424} C_VEL
LIN {X 0,Y 353.914,Z 464.805,A -85,B 0,C 180,E1 -13419.141,E2 -13419.141} C_VEL
LIN {X 0,Y 354.49,Z 458.781,A -85,B 0,C 180,E1 -13420.856,E2 -13420.856} C_VEL
LIN {X 0,Y 355.159,Z 452.684,A -85,B 0,C 180,E1 -13422.282,E2 -13422.282} C_VEL
LIN {X 0,Y 355.882,Z 446.985,A -85,B 0,C 180,E1 -13423.417,E2 -13423.417} C_VEL
LIN {X 0,Y 356.798,Z 438.429,A -85,B 0,C 180,E1 -13424.837,E2 -13424.837} C_VEL
LIN {X 0,Y 357.604,Z 430.245,A -85,B 0,C 180,E1 -13425.97,E2 -13425.97} C_VEL
LIN {X 0,Y 358.569,Z 421.735,A -85,B 0,C 180,E1 -13426.951,E2 -13426.951} C_VEL
LIN {X 0,Y 359.454,Z 413.019,A -85,B 0,C 180,E1 -13427.788,E2 -13427.788} C_VEL
LIN {X 0,Y 359.572,Z 408.111,A -85,B 0,C 180,E1 -13428.224,E2 -13428.224} C_VEL
LIN {X 0,Y 358.188,Z 396.777,A -85,B 0,C 180,E1 -13429.123,E2 -13429.123} C_VEL
LIN {X 0,Y 356.023,Z 384.598,A -85,B 0,C 180,E1 -13429.899,E2 -13429.899} C_VEL
LIN {X 0,Y 353.612,Z 373.085,A -85,B 0,C 180,E1 -13430.505,E2 -13430.505} C_VEL
LIN {X 0,Y 353.858,Z 367.696,A -85,B 0,C 180,E1 -13434.65,E2 -13434.65} C_VEL
LIN {X 0,Y 354.276,Z 362.917,A -85,B 0,C 180,E1 -13438.431,E2 -13438.431} C_VEL
LIN {X 0,Y 354.668,Z 359.103,A -85,B 0,C 180,E1 -13441.561,E2 -13441.561} C_VEL
LIN {X 0,Y 355.097,Z 355.067,A -85,B 0,C 180,E1 -13445.027,E2 -13445.027} C_VEL
LIN {X 0,Y 355.48,Z 351.976,A -85,B 0,C 180,E1 -13447.798,E2 -13447.798} C_VEL
LIN {X 0,Y 355.833,Z 348.228,A -85,B 0,C 180,E1 -13451.363,E2 -13451.363} C_VEL
LIN {X 0,Y 355.843,Z 345.904,A -85,B 0,C 180,E1 -13453.73,E2 -13453.73} C_VEL
LIN {X 0,Y 355.525,Z 342.942,A -85,B 0,C 180,E1 -13457.005,E2 -13457.005} C_VEL
LIN {X 0,Y 355.33,Z 341.08,A -85,B 0,C 180,E1 -13459.254,E2 -13459.254} C_VEL
LIN {X 0,Y 354.801,Z 337.792,A -85,B 0,C 180,E1 -13463.54,E2 -13463.54} C_VEL
LIN {X 0,Y 354.815,Z 337.788,A -85,B 0,C 180,E1 -13466.316,E2 -13466.316} C_VEL
LIN {X 0,Y 354.818,Z 337.786,A -85,B 0,C 180,E1 -13470.318,E2 -13470.318} C_VEL
LIN {X 0,Y 354.899,Z 337.776,A -85,B 0,C 180,E1 -13474.172,E2 -13474.172} C_VEL
LIN {X 0,Y 354.816,Z 337.789,A -85,B 0,C 180,E1 -13477.892,E2 -13477.892} C_VEL
LIN {X 0,Y 354.89,Z 337.778,A -85,B 0,C 180,E1 -13481.907,E2 -13481.907} C_VEL
LIN {X 0,Y 354.943,Z 337.77,A -85,B 0,C 180,E1 -13485.981,E2 -13485.981} C_VEL
LIN {X 0,Y 354.978,Z 337.767,A -85,B 0,C 180,E1 -13489.735,E2 -13489.735} C_VEL
LIN {X 0,Y 355.125,Z 337.75,A -85,B 0,C 180,E1 -13493.18,E2 -13493.18} C_VEL
LIN {X 0,Y 355.244,Z 337.732,A -85,B 0,C 180,E1 -13497.732,E2 -13497.732} C_VEL
LIN {X 0,Y 355.374,Z 337.715,A -85,B 0,C 180,E1 -13499.999,E2 -13499.999} C_VEL
LIN {X 0,Y 355.245,Z 337.73,A -85,B 0,C 180,E1 -13502.267,E2 -13502.267} C_VEL
LIN {X 0,Y 355.124,Z 337.75,A -85,B 0,C 180,E1 -13506.819,E2 -13506.819} C_VEL
LIN {X 0,Y 354.977,Z 337.765,A -85,B 0,C 180,E1 -13510.263,E2 -13510.263} C_VEL
LIN {X 0,Y 354.941,Z 337.769,A -85,B 0,C 180,E1 -13514.018,E2 -13514.018} C_VEL
LIN {X 0,Y 354.921,Z 337.772,A -85,B 0,C 180,E1 -13518.108,E2 -13518.108} C_VEL
LIN {X 0,Y 354.815,Z 337.786,A -85,B 0,C 180,E1 -13522.107,E2 -13522.107} C_VEL
LIN {X 0,Y 354.896,Z 337.775,A -85,B 0,C 180,E1 -13525.827,E2 -13525.827} C_VEL
LIN {X 0,Y 354.851,Z 337.78,A -85,B 0,C 180,E1 -13529.678,E2 -13529.678} C_VEL
LIN {X 0,Y 354.803,Z 337.787,A -85,B 0,C 180,E1 -13533.702,E2 -13533.702} C_VEL
LIN {X 0,Y 354.797,Z 337.791,A -85,B 0,C 180,E1 -13536.459,E2 -13536.459} C_VEL
LIN {X 0,Y 354.821,Z 337.784,A -85,B 0,C 180,E1 -13539.423,E2 -13539.423} C_VEL
LIN {X 0,Y 354.834,Z 337.782,A -85,B 0,C 180,E1 -13542.875,E2 -13542.875} C_VEL
LIN {X 0,Y 354.801,Z 337.792,A -85,B 0,C 180,E1 -13546.109,E2 -13546.109} C_VEL
LIN {X 0,Y 354.821,Z 337.784,A -85,B 0,C 180,E1 -13549.184,E2 -13549.184} C_VEL
LIN {X 0,Y 354.805,Z 337.787,A -85,B 0,C 180,E1 -13552.402,E2 -13552.402} C_VEL
LIN {X 0,Y 354.808,Z 337.785,A -85,B 0,C 180,E1 -13554.941,E2 -13554.941} C_VEL
LIN {X 0,Y 354.789,Z 337.788,A -85,B 0,C 180,E1 -13558.405,E2 -13558.405} C_VEL
LIN {X 0,Y 354.847,Z 337.786,A -85,B 0,C 180,E1 -13561.619,E2 -13561.619} C_VEL
LIN {X 0,Y 354.896,Z 337.776,A -85,B 0,C 180,E1 -13564.172,E2 -13564.172} C_VEL
LIN {X 0,Y 354.831,Z 337.785,A -85,B 0,C 180,E1 -13567.894,E2 -13567.894} C_VEL
LIN {X 0,Y 354.919,Z 337.776,A -85,B 0,C 180,E1 -13571.891,E2 -13571.891} C_VEL
LIN {X 0,Y 354.913,Z 337.804,A -85,B 0,C 180,E1 -13572.332,E2 -13572.332} C_VEL
LIN {X 0,Y 355.753,Z 340.372,A -85,B 0,C 180,E1 -13572.588,E2 -13572.588} C_VEL
LIN {X 0,Y 357.645,Z 342.548,A -85,B 0,C 180,E1 -13573.044,E2 -13573.044} C_VEL
LIN {X 0,Y 358.883,Z 343.495,A -85,B 0,C 180,E1 -13573.33,E2 -13573.33} C_VEL
LIN {X 0,Y 360.699,Z 346.445,A -85,B 0,C 180,E1 -13573.821,E2 -13573.821} C_VEL
LIN {X 0,Y 363.789,Z 349.336,A -85,B 0,C 180,E1 -13574.619,E2 -13574.619} C_VEL
LIN {X 0,Y 366.328,Z 352.662,A -85,B 0,C 180,E1 -13575.345,E2 -13575.345} C_VEL
LIN {X 0,Y 369.416,Z 355.28,A -85,B 0,C 180,E1 -13576.222,E2 -13576.222} C_VEL
LIN {X 0,Y 372.184,Z 358.696,A -85,B 0,C 180,E1 -13577.118,E2 -13577.118} C_VEL
LIN {X 0,Y 375.165,Z 360.964,A -85,B 0,C 180,E1 -13578.108,E2 -13578.108} C_VEL
LIN {X 0,Y 378.474,Z 364.735,A -85,B 0,C 180,E1 -13579.366,E2 -13579.366} C_VEL
LIN {X 0,Y 381.409,Z 367.009,A -85,B 0,C 180,E1 -13580.584,E2 -13580.584} C_VEL
LIN {X 0,Y 383.282,Z 368.109,A -85,B 0,C 180,E1 -13581.432,E2 -13581.432} C_VEL
LIN {X 0,Y 385.712,Z 371.138,A -85,B 0,C 180,E1 -13582.781,E2 -13582.781} C_VEL
LIN {X 0,Y 387.686,Z 372.931,A -85,B 0,C 180,E1 -13584.078,E2 -13584.078} C_VEL
LIN {X 0,Y 389.596,Z 374.12,A -85,B 0,C 180,E1 -13585.603,E2 -13585.603} C_VEL
LIN {X 0,Y 390.814,Z 374.438,A -85,B 0,C 180,E1 -13586.907,E2 -13586.907} C_VEL
LIN {X 0,Y 391.493,Z 374.612,A -85,B 0,C 180,E1 -13587.942,E2 -13587.942} C_VEL
LIN {X 0,Y 391.912,Z 374.646,A -85,B 0,C 180,E1 -13588.972,E2 -13588.972} C_VEL
LIN {X 0,Y 392.049,Z 374.672,A -85,B 0,C 180,E1 -13590,E2 -13590} C_VEL
LIN {X 0,Y 391.912,Z 374.649,A -85,B 0,C 180,E1 -13591.028,E2 -13591.028} C_VEL
LIN {X 0,Y 391.493,Z 374.605,A -85,B 0,C 180,E1 -13592.058,E2 -13592.058} C_VEL
LIN {X 0,Y 389.865,Z 374.221,A -85,B 0,C 180,E1 -13594.135,E2 -13594.135} C_VEL
LIN {X 0,Y 387.983,Z 373.15,A -85,B 0,C 180,E1 -13595.718,E2 -13595.718} C_VEL
LIN {X 0,Y 385.836,Z 371.28,A -85,B 0,C 180,E1 -13597.14,E2 -13597.14} C_VEL
LIN {X 0,Y 383.281,Z 368.111,A -85,B 0,C 180,E1 -13598.568,E2 -13598.568} C_VEL
LIN {X 0,Y 379.539,Z 365.702,A -85,B 0,C 180,E1 -13600.199,E2 -13600.199} C_VEL
LIN {X 0,Y 376.615,Z 362.711,A -85,B 0,C 180,E1 -13601.362,E2 -13601.362} C_VEL
LIN {X 0,Y 375.166,Z 360.962,A -85,B 0,C 180,E1 -13601.892,E2 -13601.892} C_VEL
LIN {X 0,Y 371.883,Z 358.4,A -85,B 0,C 180,E1 -13602.976,E2 -13602.976} C_VEL
LIN {X 0,Y 368.741,Z 354.565,A -85,B 0,C 180,E1 -13603.979,E2 -13603.979} C_VEL
LIN {X 0,Y 365.602,Z 351.886,A -85,B 0,C 180,E1 -13604.863,E2 -13604.863} C_VEL
LIN {X 0,Y 363.096,Z 348.577,A -85,B 0,C 180,E1 -13605.563,E2 -13605.563} C_VEL
LIN {X 0,Y 360.461,Z 346.159,A -85,B 0,C 180,E1 -13606.243,E2 -13606.243} C_VEL
LIN {X 0,Y 358.64,Z 343.183,A -85,B 0,C 180,E1 -13606.73,E2 -13606.73} C_VEL
LIN {X 0,Y 356.271,Z 341.19,A -85,B 0,C 180,E1 -13607.28,E2 -13607.28} C_VEL
LIN {X 0,Y 355.066,Z 338.675,A -85,B 0,C 180,E1 -13607.608,E2 -13607.608} C_VEL
LIN {X 0,Y 354.921,Z 337.776,A -85,B 0,C 180,E1 -13607.693,E2 -13607.693} C_VEL
LIN {X 0,Y 354.837,Z 337.782,A -85,B 0,C 180,E1 -13611.427,E2 -13611.427} C_VEL
LIN {X 0,Y 354.858,Z 337.784,A -85,B 0,C 180,E1 -13614.576,E2 -13614.576} C_VEL
LIN {X 0,Y 354.88,Z 337.777,A -85,B 0,C 180,E1 -13617.096,E2 -13617.096} C_VEL
LIN {X 0,Y 354.85,Z 337.781,A -85,B 0,C 180,E1 -13619.679,E2 -13619.679} C_VEL
LIN {X 0,Y 354.802,Z 337.788,A -85,B 0,C 180,E1 -13623.702,E2 -13623.702} C_VEL
LIN {X 0,Y 354.796,Z 337.789,A -85,B 0,C 180,E1 -13626.459,E2 -13626.459} C_VEL
LIN {X 0,Y 354.82,Z 337.785,A -85,B 0,C 180,E1 -13629.424,E2 -13629.424} C_VEL
LIN {X 0,Y 354.804,Z 337.786,A -85,B 0,C 180,E1 -13632.871,E2 -13632.871} C_VEL
LIN {X 0,Y 354.849,Z 337.784,A -85,B 0,C 180,E1 -13636.117,E2 -13636.117} C_VEL
LIN {X 0,Y 354.824,Z 337.781,A -85,B 0,C 180,E1 -13639.577,E2 -13639.577} C_VEL
LIN {X 0,Y 354.796,Z 337.791,A -85,B 0,C 180,E1 -13643.541,E2 -13643.541} C_VEL
LIN {X 0,Y 354.811,Z 337.785,A -85,B 0,C 180,E1 -13644.512,E2 -13644.512} C_VEL
LIN {X 0,Y 354.12,Z 337.875,A -85,B 0,C 180,E1 -13645.459,E2 -13645.459} C_VEL
LIN {X 0,Y 351.226,Z 338.232,A -85,B 0,C 180,E1 -13646.998,E2 -13646.998} C_VEL
LIN {X 0,Y 348.81,Z 338.533,A -85,B 0,C 180,E1 -13648.244,E2 -13648.244} C_VEL
LIN {X 0,Y 347.812,Z 338.659,A -85,B 0,C 180,E1 -13649.209,E2 -13649.209} C_VEL
LIN {X 0,Y 347.752,Z 338.668,A -85,B 0,C 180,E1 -13649.536,E2 -13649.536} C_VEL
LIN {X 0,Y 347.849,Z 338.653,A -85,B 0,C 180,E1 -13652.745,E2 -13652.745} C_VEL
LIN {X 0,Y 347.783,Z 338.661,A -85,B 0,C 180,E1 -13656.162,E2 -13656.162} C_VEL
LIN {X 0,Y 347.809,Z 338.658,A -85,B 0,C 180,E1 -13659.91,E2 -13659.91} C_VEL
LIN {X 0,Y 347.864,Z 338.65,A -85,B 0,C 180,E1 -13662.36,E2 -13662.36} C_VEL
LIN {X 0,Y 347.896,Z 338.646,A -85,B 0,C 180,E1 -13665.971,E2 -13665.971} C_VEL
LIN {X 0,Y 347.927,Z 338.644,A -85,B 0,C 180,E1 -13669.526,E2 -13669.526} C_VEL
LIN {X 0,Y 348.09,Z 338.628,A -85,B 0,C 180,E1 -13673.043,E2 -13673.043} C_VEL
LIN {X 0,Y 348.207,Z 338.606,A -85,B 0,C 180,E1 -13677.687,E2 -13677.687} C_VEL
LIN {X 0,Y 348.324,Z 338.592,A -85,B 0,C 180,E1 -13680.001,E2 -13680.001} C_VEL
LIN {X 0,Y 348.207,Z 338.609,A -85,B 0,C 180,E1 -13682.314,E2 -13682.314} C_VEL
LIN {X 0,Y 348.091,Z 338.625,A -85,B 0,C 180,E1 -13686.959,E2 -13686.959} C_VEL
LIN {X 0,Y 347.928,Z 338.648,A -85,B 0,C 180,E1 -13690.475,E2 -13690.475} C_VEL
LIN {X 0,Y 347.899,Z 338.649,A -85,B 0,C 180,E1 -13694.15,E2 -13694.15} C_VEL
LIN {X 0,Y 347.829,Z 338.66,A -85,B 0,C 180,E1 -13698.26,E2 -13698.26} C_VEL
LIN {X 0,Y 347.768,Z 338.663,A -85,B 0,C 180,E1 -13701.627,E2 -13701.627} C_VEL
LIN {X 0,Y 347.812,Z 338.657,A -85,B 0,C 180,E1 -13705.109,E2 -13705.109} C_VEL
LIN {X 0,Y 347.81,Z 338.659,A -85,B 0,C 180,E1 -13707.695,E2 -13707.695} C_VEL
LIN {X 0,Y 347.75,Z 338.669,A -85,B 0,C 180,E1 -13710.348,E2 -13710.348} C_VEL
LIN {X 0,Y 347.749,Z 338.671,A -85,B 0,C 180,E1 -13714.044,E2 -13714.044} C_VEL
LIN {X 0,Y 347.772,Z 338.667,A -85,B 0,C 180,E1 -13716.066,E2 -13716.066} C_VEL
LIN {X 0,Y 348.219,Z 341.737,A -85,B 0,C 180,E1 -13720.23,E2 -13720.23} C_VEL
LIN {X 0,Y 348.576,Z 344.421,A -85,B 0,C 180,E1 -13723.462,E2 -13723.462} C_VEL
LIN {X 0,Y 348.806,Z 347.134,A -85,B 0,C 180,E1 -13726.499,E2 -13726.499} C_VEL
LIN {X 0,Y 348.798,Z 348.871,A -85,B 0,C 180,E1 -13728.324,E2 -13728.324} C_VEL
LIN {X 0,Y 348.469,Z 352.492,A -85,B 0,C 180,E1 -13731.866,E2 -13731.866} C_VEL
LIN {X 0,Y 347.96,Z 356.535,A -85,B 0,C 180,E1 -13735.561,E2 -13735.561} C_VEL
LIN {X 0,Y 347.622,Z 359.652,A -85,B 0,C 180,E1 -13738.288,E2 -13738.288} C_VEL
LIN {X 0,Y 347.279,Z 362.807,A -85,B 0,C 180,E1 -13740.942,E2 -13740.942} C_VEL
LIN {X 0,Y 346.835,Z 367.559,A -85,B 0,C 180,E1 -13744.816,E2 -13744.816} C_VEL
LIN {X 0,Y 346.498,Z 372.339,A -85,B 0,C 180,E1 -13748.587,E2 -13748.587} C_VEL
LIN {X 0,Y 346.494,Z 372.943,A -85,B 0,C 180,E1 -13749.076,E2 -13749.076} C_VEL
LIN {X 0,Y 349.744,Z 388.091,A -85,B 0,C 180,E1 -13749.897,E2 -13749.897} C_VEL
LIN {X 0,Y 351.648,Z 399.807,A -85,B 0,C 180,E1 -13750.733,E2 -13750.733} C_VEL
LIN {X 0,Y 352.757,Z 409.551,A -85,B 0,C 180,E1 -13751.562,E2 -13751.562} C_VEL
LIN {X 0,Y 352.087,Z 418.836,A -85,B 0,C 180,E1 -13752.428,E2 -13752.428} C_VEL
LIN {X 0,Y 351.053,Z 427.78,A -85,B 0,C 180,E1 -13753.424,E2 -13753.424} C_VEL
LIN {X 0,Y 350.155,Z 435.528,A -85,B 0,C 180,E1 -13754.456,E2 -13754.456} C_VEL
LIN {X 0,Y 349.316,Z 443.533,A -85,B 0,C 180,E1 -13755.732,E2 -13755.732} C_VEL
LIN {X 0,Y 348.553,Z 449.736,A -85,B 0,C 180,E1 -13756.889,E2 -13756.889} C_VEL
LIN {X 0,Y 347.72,Z 456.272,A -85,B 0,C 180,E1 -13758.339,E2 -13758.339} C_VEL
LIN {X 0,Y 347.268,Z 460.776,A -85,B 0,C 180,E1 -13759.506,E2 -13759.506} C_VEL
LIN {X 0,Y 346.726,Z 466.269,A -85,B 0,C 180,E1 -13761.256,E2 -13761.256} C_VEL
LIN {X 0,Y 346.346,Z 470.594,A -85,B 0,C 180,E1 -13763.007,E2 -13763.007} C_VEL
LIN {X 0,Y 346.231,Z 472.962,A -85,B 0,C 180,E1 -13764.175,E2 -13764.175} C_VEL
LIN {X 0,Y 346.179,Z 474.762,A -85,B 0,C 180,E1 -13765.342,E2 -13765.342} C_VEL
LIN {X 0,Y 346.085,Z 477.208,A -85,B 0,C 180,E1 -13767.672,E2 -13767.672} C_VEL
LIN {X 0,Y 346.104,Z 477.797,A -85,B 0,C 180,E1 -13768.836,E2 -13768.836} C_VEL
LIN {X 0,Y 346.164,Z 477.953,A -85,B 0,C 180,E1 -13770,E2 -13770} C_VEL
LIN {X 0,Y 346.104,Z 477.797,A -85,B 0,C 180,E1 -13771.164,E2 -13771.164} C_VEL
LIN {X 0,Y 346.085,Z 477.208,A -85,B 0,C 180,E1 -13772.328,E2 -13772.328} C_VEL
LIN {X 0,Y 346.175,Z 474.762,A -85,B 0,C 180,E1 -13774.658,E2 -13774.658} C_VEL
LIN {X 0,Y 346.248,Z 471.812,A -85,B 0,C 180,E1 -13776.409,E2 -13776.409} C_VEL
LIN {X 0,Y 346.574,Z 467.823,A -85,B 0,C 180,E1 -13778.161,E2 -13778.161} C_VEL
LIN {X 0,Y 347.043,Z 462.692,A -85,B 0,C 180,E1 -13779.912,E2 -13779.912} C_VEL
LIN {X 0,Y 347.588,Z 457.428,A -85,B 0,C 180,E1 -13781.37,E2 -13781.37} C_VEL
LIN {X 0,Y 348.367,Z 451.112,A -85,B 0,C 180,E1 -13782.821,E2 -13782.821} C_VEL
LIN {X 0,Y 349.114,Z 445.161,A -85,B 0,C 180,E1 -13783.979,E2 -13783.979} C_VEL
LIN {X 0,Y 350.028,Z 437.178,A -85,B 0,C 180,E1 -13785.294,E2 -13785.294} C_VEL
LIN {X 0,Y 350.887,Z 428.914,A -85,B 0,C 180,E1 -13786.434,E2 -13786.434} C_VEL
LIN {X 0,Y 351.924,Z 420.187,A -85,B 0,C 180,E1 -13787.431,E2 -13787.431} C_VEL
LIN {X 0,Y 352.78,Z 411.189,A -85,B 0,C 180,E1 -13788.286,E2 -13788.286} C_VEL
LIN {X 0,Y 352.013,Z 402.853,A -85,B 0,C 180,E1 -13789.019,E2 -13789.019} C_VEL
LIN {X 0,Y 350.817,Z 394.155,A -85,B 0,C 180,E1 -13789.683,E2 -13789.683} C_VEL
LIN {X 0,Y 348.924,Z 383.921,A -85,B 0,C 180,E1 -13790.342,E2 -13790.342} C_VEL
LIN {X 0,Y 346.542,Z 372.916,A -85,B 0,C 180,E1 -13790.943,E2 -13790.943} C_VEL
LIN {X 0,Y 346.836,Z 367.551,A -85,B 0,C 180,E1 -13795.184,E2 -13795.184} C_VEL
LIN {X 0,Y 347.284,Z 362.795,A -85,B 0,C 180,E1 -13799.057,E2 -13799.057} C_VEL
LIN {X 0,Y 347.645,Z 359.446,A -85,B 0,C 180,E1 -13801.888,E2 -13801.888} C_VEL
LIN {X 0,Y 348.162,Z 354.981,A -85,B 0,C 180,E1 -13805.831,E2 -13805.831} C_VEL
LIN {X 0,Y 348.528,Z 351.904,A -85,B 0,C 180,E1 -13808.69,E2 -13808.69} C_VEL
LIN {X 0,Y 348.808,Z 348.746,A -85,B 0,C 180,E1 -13811.797,E2 -13811.797} C_VEL
LIN {X 0,Y 348.773,Z 345.854,A -85,B 0,C 180,E1 -13814.851,E2 -13814.851} C_VEL
LIN {X 0,Y 348.387,Z 342.919,A -85,B 0,C 180,E1 -13818.279,E2 -13818.279} C_VEL
LIN {X 0,Y 347.937,Z 340.061,A -85,B 0,C 180,E1 -13821.977,E2 -13821.977} C_VEL
LIN {X 0,Y 347.79,Z 338.667,A -85,B 0,C 180,E1 -13824.124,E2 -13824.124} C_VEL
LIN {X 0,Y 347.74,Z 338.671,A -85,B 0,C 180,E1 -13828.085,E2 -13828.085} C_VEL
LIN {X 0,Y 347.78,Z 338.661,A -85,B 0,C 180,E1 -13830.987,E2 -13830.987} C_VEL
LIN {X 0,Y 347.832,Z 338.658,A -85,B 0,C 180,E1 -13833.607,E2 -13833.607} C_VEL
LIN {X 0,Y 347.785,Z 338.663,A -85,B 0,C 180,E1 -13836.161,E2 -13836.161} C_VEL
LIN {X 0,Y 347.8,Z 338.662,A -85,B 0,C 180,E1 -13839.908,E2 -13839.908} C_VEL
LIN {X 0,Y 347.832,Z 338.66,A -85,B 0,C 180,E1 -13843.568,E2 -13843.568} C_VEL
LIN {X 0,Y 347.89,Z 338.65,A -85,B 0,C 180,E1 -13847.16,E2 -13847.16} C_VEL
LIN {X 0,Y 347.964,Z 338.638,A -85,B 0,C 180,E1 -13850.701,E2 -13850.701} C_VEL
LIN {X 0,Y 348.091,Z 338.625,A -85,B 0,C 180,E1 -13853.041,E2 -13853.041} C_VEL
LIN {X 0,Y 348.207,Z 338.609,A -85,B 0,C 180,E1 -13857.686,E2 -13857.686} C_VEL
LIN {X 0,Y 348.324,Z 338.592,A -85,B 0,C 180,E1 -13859.999,E2 -13859.999} C_VEL
LIN {X 0,Y 348.207,Z 338.606,A -85,B 0,C 180,E1 -13862.313,E2 -13862.313} C_VEL
LIN {X 0,Y 348.09,Z 338.628,A -85,B 0,C 180,E1 -13866.957,E2 -13866.957} C_VEL
LIN {X 0,Y 347.927,Z 338.644,A -85,B 0,C 180,E1 -13870.474,E2 -13870.474} C_VEL
LIN {X 0,Y 347.897,Z 338.647,A -85,B 0,C 180,E1 -13874.149,E2 -13874.149} C_VEL
LIN {X 0,Y 347.889,Z 338.649,A -85,B 0,C 180,E1 -13878.29,E2 -13878.29} C_VEL
LIN {X 0,Y 347.766,Z 338.663,A -85,B 0,C 180,E1 -13881.626,E2 -13881.626} C_VEL
LIN {X 0,Y 347.809,Z 338.658,A -85,B 0,C 180,E1 -13885.108,E2 -13885.108} C_VEL
LIN {X 0,Y 347.808,Z 338.657,A -85,B 0,C 180,E1 -13887.693,E2 -13887.693} C_VEL
LIN {X 0,Y 347.761,Z 338.668,A -85,B 0,C 180,E1 -13890.346,E2 -13890.346} C_VEL
LIN {X 0,Y 347.741,Z 338.67,A -85,B 0,C 180,E1 -13894.463,E2 -13894.463} C_VEL
LIN {X 0,Y 347.773,Z 338.665,A -85,B 0,C 180,E1 -13897.989,E2 -13897.989} C_VEL
LIN {X 0,Y 347.782,Z 338.663,A -85,B 0,C 180,E1 -13901.825,E2 -13901.825} C_VEL
LIN {X 0,Y 347.795,Z 338.659,A -85,B 0,C 180,E1 -13905.011,E2 -13905.011} C_VEL
LIN {X 0,Y 347.765,Z 338.665,A -85,B 0,C 180,E1 -13908.393,E2 -13908.393} C_VEL
LIN {X 0,Y 347.772,Z 338.667,A -85,B 0,C 180,E1 -13912.01,E2 -13912.01} C_VEL
LIN {X 0,Y 347.741,Z 338.669,A -85,B 0,C 180,E1 -13915.536,E2 -13915.536} C_VEL
LIN {X 0,Y 347.76,Z 338.669,A -85,B 0,C 180,E1 -13919.653,E2 -13919.653} C_VEL
LIN {X 0,Y 347.848,Z 338.653,A -85,B 0,C 180,E1 -13922.744,E2 -13922.744} C_VEL
LIN {X 0,Y 347.785,Z 338.662,A -85,B 0,C 180,E1 -13926.162,E2 -13926.162} C_VEL
LIN {X 0,Y 347.814,Z 338.66,A -85,B 0,C 180,E1 -13929.91,E2 -13929.91} C_VEL
LIN {X 0,Y 347.841,Z 338.658,A -85,B 0,C 180,E1 -13931.024,E2 -13931.024} C_VEL
LIN {X 0,Y 348.762,Z 341.378,A -85,B 0,C 180,E1 -13931.28,E2 -13931.28} C_VEL
LIN {X 0,Y 350.819,Z 343.568,A -85,B 0,C 180,E1 -13931.728,E2 -13931.728} C_VEL
LIN {X 0,Y 351.518,Z 344.234,A -85,B 0,C 180,E1 -13931.881,E2 -13931.881} C_VEL
LIN {X 0,Y 353.571,Z 347.401,A -85,B 0,C 180,E1 -13932.366,E2 -13932.366} C_VEL
LIN {X 0,Y 356.152,Z 350.033,A -85,B 0,C 180,E1 -13932.977,E2 -13932.977} C_VEL
LIN {X 0,Y 358.881,Z 353.477,A -85,B 0,C 180,E1 -13933.649,E2 -13933.649} C_VEL
LIN {X 0,Y 361.214,Z 355.685,A -85,B 0,C 180,E1 -13934.252,E2 -13934.252} C_VEL
LIN {X 0,Y 364.271,Z 359.231,A -85,B 0,C 180,E1 -13935.07,E2 -13935.07} C_VEL
LIN {X 0,Y 367.191,Z 361.728,A -85,B 0,C 180,E1 -13935.884,E2 -13935.884} C_VEL
LIN {X 0,Y 370.23,Z 365.267,A -85,B 0,C 180,E1 -13936.833,E2 -13936.833} C_VEL
LIN {X 0,Y 374.052,Z 368.353,A -85,B 0,C 180,E1 -13938.072,E2 -13938.072} C_VEL
LIN {X 0,Y 376.844,Z 371.446,A -85,B 0,C 180,E1 -13939.116,E2 -13939.116} C_VEL
LIN {X 0,Y 380.101,Z 373.903,A -85,B 0,C 180,E1 -13940.421,E2 -13940.421} C_VEL
LIN {X 0,Y 382.04,Z 375.159,A -85,B 0,C 180,E1 -13941.287,E2 -13941.287} C_VEL
LIN {X 0,Y 384.762,Z 378.339,A -85,B 0,C 180,E1 -13942.763,E2 -13942.763} C_VEL
LIN {X 0,Y 387.068,Z 380.227,A -85,B 0,C 180,E1 -13944.269,E2 -13944.269} C_VEL
LIN {X 0,Y 388.979,Z 381.243,A -85,B 0,C 180,E1 -13945.856,E2 -13945.856} C_VEL
LIN {X 0,Y 389.939,Z 381.471,A -85,B 0,C 180,E1 -13946.901,E2 -13946.901} C_VEL
LIN {X 0,Y 390.625,Z 381.629,A -85,B 0,C 180,E1 -13947.938,E2 -13947.938} C_VEL
LIN {X 0,Y 391.046,Z 381.674,A -85,B 0,C 180,E1 -13948.97,E2 -13948.97} C_VEL
LIN {X 0,Y 391.184,Z 381.718,A -85,B 0,C 180,E1 -13950,E2 -13950} C_VEL
LIN {X 0,Y 391.046,Z 381.678,A -85,B 0,C 180,E1 -13951.03,E2 -13951.03} C_VEL
LIN {X 0,Y 390.621,Z 381.65,A -85,B 0,C 180,E1 -13952.062,E2 -13952.062} C_VEL
LIN {X 0,Y 389.525,Z 381.372,A -85,B 0,C 180,E1 -13953.61,E2 -13953.61} C_VEL
LIN {X 0,Y 387.766,Z 380.674,A -85,B 0,C 180,E1 -13955.199,E2 -13955.199} C_VEL
LIN {X 0,Y 385.509,Z 379.052,A -85,B 0,C 180,E1 -13956.768,E2 -13956.768} C_VEL
LIN {X 0,Y 382.72,Z 376.05,A -85,B 0,C 180,E1 -13958.361,E2 -13958.361} C_VEL
LIN {X 0,Y 381.489,Z 374.605,A -85,B 0,C 180,E1 -13958.984,E2 -13958.984} C_VEL
LIN {X 0,Y 378.16,Z 372.577,A -85,B 0,C 180,E1 -13960.372,E2 -13960.372} C_VEL
LIN {X 0,Y 374.823,Z 369.37,A -85,B 0,C 180,E1 -13961.64,E2 -13961.64} C_VEL
LIN {X 0,Y 373.241,Z 367.578,A -85,B 0,C 180,E1 -13962.213,E2 -13962.213} C_VEL
LIN {X 0,Y 369.642,Z 364.683,A -85,B 0,C 180,E1 -13963.353,E2 -13963.353} C_VEL
LIN {X 0,Y 366.192,Z 360.78,A -85,B 0,C 180,E1 -13964.4,E2 -13964.4} C_VEL
LIN {X 0,Y 362.952,Z 357.925,A -85,B 0,C 180,E1 -13965.278,E2 -13965.278} C_VEL
LIN {X 0,Y 360.503,Z 354.851,A -85,B 0,C 180,E1 -13965.94,E2 -13965.94} C_VEL
LIN {X 0,Y 357.57,Z 352.063,A -85,B 0,C 180,E1 -13966.664,E2 -13966.664} C_VEL
LIN {X 0,Y 355.395,Z 349.095,A -85,B 0,C 180,E1 -13967.209,E2 -13967.209} C_VEL
LIN {X 0,Y 352.737,Z 346.376,A -85,B 0,C 180,E1 -13967.823,E2 -13967.823} C_VEL
LIN {X 0,Y 351.387,Z 343.913,A -85,B 0,C 180,E1 -13968.154,E2 -13968.154} C_VEL
LIN {X 0,Y 349.085,Z 341.869,A -85,B 0,C 180,E1 -13968.645,E2 -13968.645} C_VEL
LIN {X 0,Y 347.946,Z 339.334,A -85,B 0,C 180,E1 -13968.932,E2 -13968.932} C_VEL
LIN {X 0,Y 347.829,Z 338.66,A -85,B 0,C 180,E1 -13969.015,E2 -13969.015} C_VEL
LIN {X 0,Y 347.771,Z 338.667,A -85,B 0,C 180,E1 -13972.579,E2 -13972.579} C_VEL
LIN {X 0,Y 347.808,Z 338.658,A -85,B 0,C 180,E1 -13975.109,E2 -13975.109} C_VEL
LIN {X 0,Y 347.807,Z 338.658,A -85,B 0,C 180,E1 -13977.694,E2 -13977.694} C_VEL
LIN {X 0,Y 347.76,Z 338.669,A -85,B 0,C 180,E1 -13980.347,E2 -13980.347} C_VEL
LIN {X 0,Y 347.741,Z 338.669,A -85,B 0,C 180,E1 -13984.464,E2 -13984.464} C_VEL
LIN {X 0,Y 347.772,Z 338.667,A -85,B 0,C 180,E1 -13987.99,E2 -13987.99} C_VEL
LIN {X 0,Y 347.763,Z 338.667,A -85,B 0,C 180,E1 -13991.828,E2 -13991.828} C_VEL
LIN {X 0,Y 347.795,Z 338.659,A -85,B 0,C 180,E1 -13995.012,E2 -13995.012} C_VEL
LIN {X 0,Y 347.783,Z 338.662,A -85,B 0,C 180,E1 -13998.391,E2 -13998.391} C_VEL
LIN {X 0,Y 347.773,Z 338.665,A -85,B 0,C 180,E1 -14002.011,E2 -14002.011} C_VEL
LIN {X 0,Y 347.741,Z 338.67,A -85,B 0,C 180,E1 -14005.537,E2 -14005.537} C_VEL
LIN {X 0,Y 347.752,Z 338.668,A -85,B 0,C 180,E1 -14009.536,E2 -14009.536} C_VEL
LIN {X 0,Y 347.143,Z 338.75,A -85,B 0,C 180,E1 -14010.503,E2 -14010.503} C_VEL
LIN {X 0,Y 344.321,Z 339.1,A -85,B 0,C 180,E1 -14012.078,E2 -14012.078} C_VEL
LIN {X 0,Y 341.894,Z 339.399,A -85,B 0,C 180,E1 -14013.353,E2 -14013.353} C_VEL
LIN {X 0,Y 340.845,Z 339.525,A -85,B 0,C 180,E1 -14014.339,E2 -14014.339} C_VEL
LIN {X 0,Y 340.758,Z 339.535,A -85,B 0,C 180,E1 -14014.673,E2 -14014.673} C_VEL
LIN {X 0,Y 340.739,Z 339.538,A -85,B 0,C 180,E1 -14018.207,E2 -14018.207} C_VEL
LIN {X 0,Y 340.856,Z 339.524,A -85,B 0,C 180,E1 -14021.985,E2 -14021.985} C_VEL
LIN {X 0,Y 340.868,Z 339.523,A -85,B 0,C 180,E1 -14025.706,E2 -14025.706} C_VEL
LIN {X 0,Y 340.869,Z 339.525,A -85,B 0,C 180,E1 -14029.307,E2 -14029.307} C_VEL
LIN {X 0,Y 341.059,Z 339.503,A -85,B 0,C 180,E1 -14032.899,E2 -14032.899} C_VEL
LIN {X 0,Y 341.169,Z 339.482,A -85,B 0,C 180,E1 -14037.639,E2 -14037.639} C_VEL
LIN {X 0,Y 341.275,Z 339.47,A -85,B 0,C 180,E1 -14040.001,E2 -14040.001} C_VEL
LIN {X 0,Y 341.169,Z 339.486,A -85,B 0,C 180,E1 -14042.362,E2 -14042.362} C_VEL
LIN {X 0,Y 341.059,Z 339.5,A -85,B 0,C 180,E1 -14047.103,E2 -14047.103} C_VEL
LIN {X 0,Y 340.871,Z 339.526,A -85,B 0,C 180,E1 -14050.694,E2 -14050.694} C_VEL
LIN {X 0,Y 340.863,Z 339.527,A -85,B 0,C 180,E1 -14054.325,E2 -14054.325} C_VEL
LIN {X 0,Y 340.786,Z 339.538,A -85,B 0,C 180,E1 -14058.441,E2 -14058.441} C_VEL
LIN {X 0,Y 340.718,Z 339.543,A -85,B 0,C 180,E1 -14061.842,E2 -14061.842} C_VEL
LIN {X 0,Y 340.773,Z 339.536,A -85,B 0,C 180,E1 -14065.665,E2 -14065.665} C_VEL
LIN {X 0,Y 340.73,Z 339.544,A -85,B 0,C 180,E1 -14068.321,E2 -14068.321} C_VEL
LIN {X 0,Y 340.699,Z 339.544,A -85,B 0,C 180,E1 -14071.045,E2 -14071.045} C_VEL
LIN {X 0,Y 340.719,Z 339.544,A -85,B 0,C 180,E1 -14075.279,E2 -14075.279} C_VEL
LIN {X 0,Y 340.812,Z 340.225,A -85,B 0,C 180,E1 -14076.729,E2 -14076.729} C_VEL
LIN {X 0,Y 341.211,Z 342.916,A -85,B 0,C 180,E1 -14080.351,E2 -14080.351} C_VEL
LIN {X 0,Y 341.593,Z 345.87,A -85,B 0,C 180,E1 -14083.938,E2 -14083.938} C_VEL
LIN {X 0,Y 341.756,Z 347.678,A -85,B 0,C 180,E1 -14086.035,E2 -14086.035} C_VEL
LIN {X 0,Y 341.7,Z 350.319,A -85,B 0,C 180,E1 -14088.84,E2 -14088.84} C_VEL
LIN {X 0,Y 341.415,Z 353.365,A -85,B 0,C 180,E1 -14091.863,E2 -14091.863} C_VEL
LIN {X 0,Y 340.908,Z 357.304,A -85,B 0,C 180,E1 -14095.551,E2 -14095.551} C_VEL
LIN {X 0,Y 340.456,Z 361.108,A -85,B 0,C 180,E1 -14098.931,E2 -14098.931} C_VEL
LIN {X 0,Y 339.952,Z 365.59,A -85,B 0,C 180,E1 -14102.744,E2 -14102.744} C_VEL
LIN {X 0,Y 339.699,Z 369.022,A -85,B 0,C 180,E1 -14105.558,E2 -14105.558} C_VEL
LIN {X 0,Y 339.41,Z 372.782,A -85,B 0,C 180,E1 -14108.625,E2 -14108.625} C_VEL
LIN {X 0,Y 342.556,Z 386.877,A -85,B 0,C 180,E1 -14109.404,E2 -14109.404} C_VEL
LIN {X 0,Y 344.694,Z 399.451,A -85,B 0,C 180,E1 -14110.316,E2 -14110.316} C_VEL
LIN {X 0,Y 345.803,Z 409.349,A -85,B 0,C 180,E1 -14111.178,E2 -14111.178} C_VEL
LIN {X 0,Y 345.779,Z 414.259,A -85,B 0,C 180,E1 -14111.637,E2 -14111.637} C_VEL
LIN {X 0,Y 344.393,Z 426.449,A -85,B 0,C 180,E1 -14112.941,E2 -14112.941} C_VEL
LIN {X 0,Y 343.432,Z 434.511,A -85,B 0,C 180,E1 -14114.013,E2 -14114.013} C_VEL
LIN {X 0,Y 342.374,Z 443.336,A -85,B 0,C 180,E1 -14115.436,E2 -14115.436} C_VEL
LIN {X 0,Y 341.622,Z 449.539,A -85,B 0,C 180,E1 -14116.618,E2 -14116.618} C_VEL
LIN {X 0,Y 340.74,Z 456.076,A -85,B 0,C 180,E1 -14118.097,E2 -14118.097} C_VEL
LIN {X 0,Y 340.255,Z 460.579,A -85,B 0,C 180,E1 -14119.287,E2 -14119.287} C_VEL
LIN {X 0,Y 339.69,Z 466.073,A -85,B 0,C 180,E1 -14121.073,E2 -14121.073} C_VEL
LIN {X 0,Y 339.277,Z 470.398,A -85,B 0,C 180,E1 -14122.86,E2 -14122.86} C_VEL
LIN {X 0,Y 339.137,Z 472.854,A -85,B 0,C 180,E1 -14124.11,E2 -14124.11} C_VEL
LIN {X 0,Y 339.072,Z 475.955,A -85,B 0,C 180,E1 -14126.435,E2 -14126.435} C_VEL
LIN {X 0,Y 338.999,Z 477.012,A -85,B 0,C 180,E1 -14127.624,E2 -14127.624} C_VEL
LIN {X 0,Y 339.007,Z 477.601,A -85,B 0,C 180,E1 -14128.812,E2 -14128.812} C_VEL
LIN {X 0,Y 339.066,Z 477.757,A -85,B 0,C 180,E1 -14130,E2 -14130} C_VEL
LIN {X 0,Y 339.007,Z 477.601,A -85,B 0,C 180,E1 -14131.188,E2 -14131.188} C_VEL
LIN {X 0,Y 338.999,Z 477.012,A -85,B 0,C 180,E1 -14132.376,E2 -14132.376} C_VEL
LIN {X 0,Y 339.076,Z 474.566,A -85,B 0,C 180,E1 -14134.756,E2 -14134.756} C_VEL
LIN {X 0,Y 339.17,Z 471.614,A -85,B 0,C 180,E1 -14136.544,E2 -14136.544} C_VEL
LIN {X 0,Y 339.534,Z 467.627,A -85,B 0,C 180,E1 -14138.331,E2 -14138.331} C_VEL
LIN {X 0,Y 340.037,Z 462.496,A -85,B 0,C 180,E1 -14140.118,E2 -14140.118} C_VEL
LIN {X 0,Y 340.594,Z 457.231,A -85,B 0,C 180,E1 -14141.606,E2 -14141.606} C_VEL
LIN {X 0,Y 341.421,Z 450.915,A -85,B 0,C 180,E1 -14143.087,E2 -14143.087} C_VEL
LIN {X 0,Y 342.182,Z 444.963,A -85,B 0,C 180,E1 -14144.268,E2 -14144.268} C_VEL
LIN {X 0,Y 343.039,Z 438.036,A -85,B 0,C 180,E1 -14145.446,E2 -14145.446} C_VEL
LIN {X 0,Y 343.912,Z 429.852,A -85,B 0,C 180,E1 -14146.624,E2 -14146.624} C_VEL
LIN {X 0,Y 344.987,Z 421.343,A -85,B 0,C 180,E1 -14147.64,E2 -14147.64} C_VEL
LIN {X 0,Y 345.901,Z 412.625,A -85,B 0,C 180,E1 -14148.51,E2 -14148.51} C_VEL
LIN {X 0,Y 345.294,Z 404.527,A -85,B 0,C 180,E1 -14149.261,E2 -14149.261} C_VEL
LIN {X 0,Y 344.054,Z 395.278,A -85,B 0,C 180,E1 -14150.007,E2 -14150.007} C_VEL
LIN {X 0,Y 342.005,Z 384.157,A -85,B 0,C 180,E1 -14150.752,E2 -14150.752} C_VEL
LIN {X 0,Y 339.446,Z 372.785,A -85,B 0,C 180,E1 -14151.371,E2 -14151.371} C_VEL
LIN {X 0,Y 339.806,Z 367.405,A -85,B 0,C 180,E1 -14155.743,E2 -14155.743} C_VEL
LIN {X 0,Y 340.32,Z 362.514,A -85,B 0,C 180,E1 -14159.847,E2 -14159.847} C_VEL
LIN {X 0,Y 340.812,Z 357.982,A -85,B 0,C 180,E1 -14163.833,E2 -14163.833} C_VEL
LIN {X 0,Y 341.203,Z 354.892,A -85,B 0,C 180,E1 -14166.679,E2 -14166.679} C_VEL
LIN {X 0,Y 341.547,Z 351.833,A -85,B 0,C 180,E1 -14169.634,E2 -14169.634} C_VEL
LIN {X 0,Y 341.76,Z 348.802,A -85,B 0,C 180,E1 -14172.735,E2 -14172.735} C_VEL
LIN {X 0,Y 341.628,Z 346.195,A -85,B 0,C 180,E1 -14175.616,E2 -14175.616} C_VEL
LIN {X 0,Y 341.29,Z 343.569,A -85,B 0,C 180,E1 -14178.779,E2 -14178.779} C_VEL
LIN {X 0,Y 340.94,Z 341.29,A -85,B 0,C 180,E1 -14181.799,E2 -14181.799} C_VEL
LIN {X 0,Y 340.794,Z 340.035,A -85,B 0,C 180,E1 -14183.54,E2 -14183.54} C_VEL
LIN {X 0,Y 340.719,Z 339.549,A -85,B 0,C 180,E1 -14184.721,E2 -14184.721} C_VEL
LIN {X 0,Y 340.699,Z 339.544,A -85,B 0,C 180,E1 -14188.955,E2 -14188.955} C_VEL
LIN {X 0,Y 340.805,Z 339.53,A -85,B 0,C 180,E1 -14193.019,E2 -14193.019} C_VEL
LIN {X 0,Y 340.755,Z 339.541,A -85,B 0,C 180,E1 -14195.638,E2 -14195.638} C_VEL
LIN {X 0,Y 340.731,Z 339.543,A -85,B 0,C 180,E1 -14199.473,E2 -14199.473} C_VEL
LIN {X 0,Y 340.792,Z 339.534,A -85,B 0,C 180,E1 -14201.98,E2 -14201.98} C_VEL
LIN {X 0,Y 340.869,Z 339.526,A -85,B 0,C 180,E1 -14205.704,E2 -14205.704} C_VEL
LIN {X 0,Y 340.871,Z 339.526,A -85,B 0,C 180,E1 -14209.306,E2 -14209.306} C_VEL
LIN {X 0,Y 341.059,Z 339.5,A -85,B 0,C 180,E1 -14212.897,E2 -14212.897} C_VEL
LIN {X 0,Y 341.169,Z 339.486,A -85,B 0,C 180,E1 -14217.638,E2 -14217.638} C_VEL
LIN {X 0,Y 341.275,Z 339.47,A -85,B 0,C 180,E1 -14219.999,E2 -14219.999} C_VEL
LIN {X 0,Y 341.169,Z 339.482,A -85,B 0,C 180,E1 -14222.361,E2 -14222.361} C_VEL
LIN {X 0,Y 341.059,Z 339.503,A -85,B 0,C 180,E1 -14227.101,E2 -14227.101} C_VEL
LIN {X 0,Y 340.869,Z 339.525,A -85,B 0,C 180,E1 -14230.693,E2 -14230.693} C_VEL
LIN {X 0,Y 340.861,Z 339.524,A -85,B 0,C 180,E1 -14234.324,E2 -14234.324} C_VEL
LIN {X 0,Y 340.836,Z 339.529,A -85,B 0,C 180,E1 -14238.466,E2 -14238.466} C_VEL
LIN {X 0,Y 340.715,Z 339.541,A -85,B 0,C 180,E1 -14241.841,E2 -14241.841} C_VEL
LIN {X 0,Y 340.77,Z 339.534,A -85,B 0,C 180,E1 -14245.664,E2 -14245.664} C_VEL
LIN {X 0,Y 340.738,Z 339.542,A -85,B 0,C 180,E1 -14248.319,E2 -14248.319} C_VEL
LIN {X 0,Y 340.702,Z 339.543,A -85,B 0,C 180,E1 -14251.043,E2 -14251.043} C_VEL
LIN {X 0,Y 340.715,Z 339.541,A -85,B 0,C 180,E1 -14255.278,E2 -14255.278} C_VEL
LIN {X 0,Y 340.715,Z 339.546,A -85,B 0,C 180,E1 -14258.387,E2 -14258.387} C_VEL
LIN {X 0,Y 340.723,Z 339.54,A -85,B 0,C 180,E1 -14261.303,E2 -14261.303} C_VEL
LIN {X 0,Y 340.735,Z 339.54,A -85,B 0,C 180,E1 -14264.529,E2 -14264.529} C_VEL
LIN {X 0,Y 340.73,Z 339.544,A -85,B 0,C 180,E1 -14267.948,E2 -14267.948} C_VEL
LIN {X 0,Y 340.735,Z 339.543,A -85,B 0,C 180,E1 -14271.773,E2 -14271.773} C_VEL
LIN {X 0,Y 340.719,Z 339.544,A -85,B 0,C 180,E1 -14275.595,E2 -14275.595} C_VEL
LIN {X 0,Y 340.7,Z 339.543,A -85,B 0,C 180,E1 -14278.956,E2 -14278.956} C_VEL
LIN {X 0,Y 340.775,Z 339.534,A -85,B 0,C 180,E1 -14282.474,E2 -14282.474} C_VEL
LIN {X 0,Y 340.752,Z 339.542,A -85,B 0,C 180,E1 -14285.638,E2 -14285.638} C_VEL
LIN {X 0,Y 340.78,Z 339.538,A -85,B 0,C 180,E1 -14289.76,E2 -14289.76} C_VEL
LIN {X 0,Y 340.825,Z 339.888,A -85,B 0,C 180,E1 -14289.869,E2 -14289.869} C_VEL
LIN {X 0,Y 341.842,Z 342.504,A -85,B 0,C 180,E1 -14290.115,E2 -14290.115} C_VEL
LIN {X 0,Y 344.233,Z 345.148,A -85,B 0,C 180,E1 -14290.594,E2 -14290.594} C_VEL
LIN {X 0,Y 346.497,Z 348.404,A -85,B 0,C 180,E1 -14291.08,E2 -14291.08} C_VEL
LIN {X 0,Y 348.434,Z 350.483,A -85,B 0,C 180,E1 -14291.493,E2 -14291.493} C_VEL
LIN {X 0,Y 351.188,Z 354.058,A -85,B 0,C 180,E1 -14292.122,E2 -14292.122} C_VEL
LIN {X 0,Y 353.192,Z 356.03,A -85,B 0,C 180,E1 -14292.56,E2 -14292.56} C_VEL
LIN {X 0,Y 356.395,Z 359.826,A -85,B 0,C 180,E1 -14293.344,E2 -14293.344} C_VEL
LIN {X 0,Y 358.763,Z 362.069,A -85,B 0,C 180,E1 -14293.91,E2 -14293.91} C_VEL
LIN {X 0,Y 361.955,Z 365.623,A -85,B 0,C 180,E1 -14294.759,E2 -14294.759} C_VEL
LIN {X 0,Y 365.023,Z 368.351,A -85,B 0,C 180,E1 -14295.582,E2 -14295.582} C_VEL
LIN {X 0,Y 368.61,Z 372.155,A -85,B 0,C 180,E1 -14296.65,E2 -14296.65} C_VEL
LIN {X 0,Y 372.227,Z 375.015,A -85,B 0,C 180,E1 -14297.794,E2 -14297.794} C_VEL
LIN {X 0,Y 375.359,Z 378.323,A -85,B 0,C 180,E1 -14298.935,E2 -14298.935} C_VEL
LIN {X 0,Y 378.786,Z 380.798,A -85,B 0,C 180,E1 -14300.286,E2 -14300.286} C_VEL
LIN {X 0,Y 380.644,Z 382.059,A -85,B 0,C 180,E1 -14301.105,E2 -14301.105} C_VEL
LIN {X 0,Y 383.3,Z 385.145,A -85,B 0,C 180,E1 -14302.555,E2 -14302.555} C_VEL
LIN {X 0,Y 385.744,Z 387.128,A -85,B 0,C 180,E1 -14304.118,E2 -14304.118} C_VEL
LIN {X 0,Y 387.876,Z 388.255,A -85,B 0,C 180,E1 -14305.844,E2 -14305.844} C_VEL
LIN {X 0,Y 388.851,Z 388.487,A -85,B 0,C 180,E1 -14306.892,E2 -14306.892} C_VEL
LIN {X 0,Y 389.956,Z 388.669,A -85,B 0,C 180,E1 -14308.967,E2 -14308.967} C_VEL
LIN {X 0,Y 390.099,Z 388.734,A -85,B 0,C 180,E1 -14310,E2 -14310} C_VEL
LIN {X 0,Y 389.956,Z 388.669,A -85,B 0,C 180,E1 -14311.033,E2 -14311.033} C_VEL
LIN {X 0,Y 389.525,Z 388.662,A -85,B 0,C 180,E1 -14312.068,E2 -14312.068} C_VEL
LIN {X 0,Y 388.406,Z 388.374,A -85,B 0,C 180,E1 -14313.62,E2 -14313.62} C_VEL
LIN {X 0,Y 386.643,Z 387.689,A -85,B 0,C 180,E1 -14315.214,E2 -14315.214} C_VEL
LIN {X 0,Y 384.078,Z 385.849,A -85,B 0,C 180,E1 -14316.986,E2 -14316.986} C_VEL
LIN {X 0,Y 381.302,Z 382.919,A -85,B 0,C 180,E1 -14318.546,E2 -14318.546} C_VEL
LIN {X 0,Y 380.047,Z 381.471,A -85,B 0,C 180,E1 -14319.169,E2 -14319.169} C_VEL
LIN {X 0,Y 376.501,Z 379.266,A -85,B 0,C 180,E1 -14320.631,E2 -14320.631} C_VEL
LIN {X 0,Y 372.918,Z 375.876,A -85,B 0,C 180,E1 -14321.964,E2 -14321.964} C_VEL
LIN {X 0,Y 371.191,Z 374.072,A -85,B 0,C 180,E1 -14322.549,E2 -14322.549} C_VEL
LIN {X 0,Y 367.554,Z 371.159,A -85,B 0,C 180,E1 -14323.67,E2 -14323.67} C_VEL
LIN {X 0,Y 363.73,Z 367.058,A -85,B 0,C 180,E1 -14324.784,E2 -14324.784} C_VEL
LIN {X 0,Y 360.112,Z 363.815,A -85,B 0,C 180,E1 -14325.721,E2 -14325.721} C_VEL
LIN {X 0,Y 357.641,Z 360.863,A -85,B 0,C 180,E1 -14326.368,E2 -14326.368} C_VEL
LIN {X 0,Y 354.116,Z 357.352,A -85,B 0,C 180,E1 -14327.209,E2 -14327.209} C_VEL
LIN {X 0,Y 352.211,Z 354.967,A -85,B 0,C 180,E1 -14327.657,E2 -14327.657} C_VEL
LIN {X 0,Y 349.106,Z 351.55,A -85,B 0,C 180,E1 -14328.35,E2 -14328.35} C_VEL
LIN {X 0,Y 347.586,Z 349.427,A -85,B 0,C 180,E1 -14328.694,E2 -14328.694} C_VEL
LIN {X 0,Y 344.987,Z 346.499,A -85,B 0,C 180,E1 -14329.238,E2 -14329.238} C_VEL
LIN {X 0,Y 343.718,Z 344.458,A -85,B 0,C 180,E1 -14329.512,E2 -14329.512} C_VEL
LIN {X 0,Y 341.672,Z 342.221,A -85,B 0,C 180,E1 -14329.922,E2 -14329.922} C_VEL
LIN {X 0,Y 340.774,Z 339.538,A -85,B 0,C 180,E1 -14330.188,E2 -14330.188} C_VEL
LIN {X 0,Y 340.725,Z 339.541,A -85,B 0,C 180,E1 -14333.073,E2 -14333.073} C_VEL
LIN {X 0,Y 340.801,Z 339.531,A -85,B 0,C 180,E1 -14336.98,E2 -14336.98} C_VEL
LIN {X 0,Y 340.759,Z 339.539,A -85,B 0,C 180,E1 -14339.978,E2 -14339.978} C_VEL
LIN {X 0,Y 340.69,Z 339.547,A -85,B 0,C 180,E1 -14343.847,E2 -14343.847} C_VEL
LIN {X 0,Y 340.702,Z 339.543,A -85,B 0,C 180,E1 -14346.742,E2 -14346.742} C_VEL
LIN {X 0,Y 340.706,Z 339.546,A -85,B 0,C 180,E1 -14350.252,E2 -14350.252} C_VEL
LIN {X 0,Y 340.704,Z 339.547,A -85,B 0,C 180,E1 -14353.783,E2 -14353.783} C_VEL
LIN {X 0,Y 340.738,Z 339.538,A -85,B 0,C 180,E1 -14357.106,E2 -14357.106} C_VEL
LIN {X 0,Y 340.731,Z 339.541,A -85,B 0,C 180,E1 -14360.253,E2 -14360.253} C_VEL
LIN {X 0,Y 340.708,Z 339.546,A -85,B 0,C 180,E1 -14363.56,E2 -14363.56} C_VEL
LIN {X 0,Y 340.691,Z 339.545,A -85,B 0,C 180,E1 -14366.154,E2 -14366.154} C_VEL
LIN {X 0,Y 340.772,Z 339.534,A -85,B 0,C 180,E1 -14370.333,E2 -14370.333} C_VEL
LIN {X 0,Y 340.802,Z 339.532,A -85,B 0,C 180,E1 -14373.021,E2 -14373.021} C_VEL
LIN {X 0,Y 340.758,Z 339.535,A -85,B 0,C 180,E1 -14374.673,E2 -14374.673} C_VEL
LIN {X 0,Y 340.074,Z 339.625,A -85,B 0,C 180,E1 -14375.66,E2 -14375.66} C_VEL
LIN {X 0,Y 337.177,Z 339.986,A -85,B 0,C 180,E1 -14377.264,E2 -14377.264} C_VEL
LIN {X 0,Y 334.756,Z 340.284,A -85,B 0,C 180,E1 -14378.563,E2 -14378.563} C_VEL
LIN {X 0,Y 333.756,Z 340.41,A -85,B 0,C 180,E1 -14379.569,E2 -14379.569} C_VEL
LIN {X 0,Y 333.696,Z 340.413,A -85,B 0,C 180,E1 -14379.91,E2 -14379.91} C_VEL
LIN {X 0,Y 333.745,Z 340.412,A -85,B 0,C 180,E1 -14382.854,E2 -14382.854} C_VEL
LIN {X 0,Y 333.795,Z 340.404,A -85,B 0,C 180,E1 -14386.609,E2 -14386.609} C_VEL
LIN {X 0,Y 333.859,Z 340.394,A -85,B 0,C 180,E1 -14390.306,E2 -14390.306} C_VEL
LIN {X 0,Y 334.011,Z 340.379,A -85,B 0,C 180,E1 -14392.748,E2 -14392.748} C_VEL
LIN {X 0,Y 333.808,Z 340.403,A -85,B 0,C 180,E1 -14395.17,E2 -14395.17} C_VEL
LIN {X 0,Y 334.106,Z 340.36,A -85,B 0,C 180,E1 -14397.589,E2 -14397.589} C_VEL
LIN {X 0,Y 334.227,Z 340.347,A -85,B 0,C 180,E1 -14400.001,E2 -14400.001} C_VEL
LIN {X 0,Y 334.106,Z 340.366,A -85,B 0,C 180,E1 -14402.412,E2 -14402.412} C_VEL
LIN {X 0,Y 334.014,Z 340.377,A -85,B 0,C 180,E1 -14406.04,E2 -14406.04} C_VEL
LIN {X 0,Y 333.984,Z 340.384,A -85,B 0,C 180,E1 -14408.502,E2 -14408.502} C_VEL
LIN {X 0,Y 333.792,Z 340.406,A -85,B 0,C 180,E1 -14412.155,E2 -14412.155} C_VEL
LIN {X 0,Y 333.808,Z 340.406,A -85,B 0,C 180,E1 -14414.635,E2 -14414.635} C_VEL
LIN {X 0,Y 333.753,Z 340.412,A -85,B 0,C 180,E1 -14418.633,E2 -14418.633} C_VEL
LIN {X 0,Y 333.657,Z 340.426,A -85,B 0,C 180,E1 -14422.281,E2 -14422.281} C_VEL
LIN {X 0,Y 333.736,Z 340.416,A -85,B 0,C 180,E1 -14426.247,E2 -14426.247} C_VEL
LIN {X 0,Y 333.691,Z 340.417,A -85,B 0,C 180,E1 -14428.975,E2 -14428.975} C_VEL
LIN {X 0,Y 333.644,Z 340.426,A -85,B 0,C 180,E1 -14432.588,E2 -14432.588} C_VEL
LIN {X 0,Y 333.687,Z 340.421,A -85,B 0,C 180,E1 -14434.775,E2 -14434.775} C_VEL
LIN {X 0,Y 333.804,Z 341.441,A -85,B 0,C 180,E1 -14436.864,E2 -14436.864} C_VEL
LIN {X 0,Y 334.253,Z 344.361,A -85,B 0,C 180,E1 -14440.805,E2 -14440.805} C_VEL
LIN {X 0,Y 334.607,Z 347.263,A -85,B 0,C 180,E1 -14444.429,E2 -14444.429} C_VEL
LIN {X 0,Y 334.724,Z 350.256,A -85,B 0,C 180,E1 -14447.788,E2 -14447.788} C_VEL
LIN {X 0,Y 334.443,Z 353.393,A -85,B 0,C 180,E1 -14451.035,E2 -14451.035} C_VEL
LIN {X 0,Y 334.057,Z 356.341,A -85,B 0,C 180,E1 -14453.909,E2 -14453.909} C_VEL
LIN {X 0,Y 333.566,Z 360.135,A -85,B 0,C 180,E1 -14457.435,E2 -14457.435} C_VEL
LIN {X 0,Y 333.091,Z 364.118,A -85,B 0,C 180,E1 -14460.969,E2 -14460.969} C_VEL
LIN {X 0,Y 332.635,Z 369.205,A -85,B 0,C 180,E1 -14465.302,E2 -14465.302} C_VEL
LIN {X 0,Y 332.385,Z 372.699,A -85,B 0,C 180,E1 -14468.168,E2 -14468.168} C_VEL
LIN {X 0,Y 334.465,Z 381.593,A -85,B 0,C 180,E1 -14468.649,E2 -14468.649} C_VEL
LIN {X 0,Y 336.145,Z 389.865,A -85,B 0,C 180,E1 -14469.18,E2 -14469.18} C_VEL
LIN {X 0,Y 337.803,Z 400.004,A -85,B 0,C 180,E1 -14469.957,E2 -14469.957} C_VEL
LIN {X 0,Y 338.875,Z 409.147,A -85,B 0,C 180,E1 -14470.778,E2 -14470.778} C_VEL
LIN {X 0,Y 339.033,Z 414.062,A -85,B 0,C 180,E1 -14471.258,E2 -14471.258} C_VEL
LIN {X 0,Y 337.598,Z 426.253,A -85,B 0,C 180,E1 -14472.587,E2 -14472.587} C_VEL
LIN {X 0,Y 336.599,Z 434.002,A -85,B 0,C 180,E1 -14473.629,E2 -14473.629} C_VEL
LIN {X 0,Y 335.464,Z 443.139,A -85,B 0,C 180,E1 -14475.129,E2 -14475.129} C_VEL
LIN {X 0,Y 334.704,Z 449.343,A -85,B 0,C 180,E1 -14476.336,E2 -14476.336} C_VEL
LIN {X 0,Y 333.759,Z 455.879,A -85,B 0,C 180,E1 -14477.844,E2 -14477.844} C_VEL
LIN {X 0,Y 333.248,Z 460.383,A -85,B 0,C 180,E1 -14479.059,E2 -14479.059} C_VEL
LIN {X 0,Y 332.635,Z 465.876,A -85,B 0,C 180,E1 -14480.882,E2 -14480.882} C_VEL
LIN {X 0,Y 332.204,Z 470.201,A -85,B 0,C 180,E1 -14482.708,E2 -14482.708} C_VEL
LIN {X 0,Y 332.038,Z 472.929,A -85,B 0,C 180,E1 -14484.167,E2 -14484.167} C_VEL
LIN {X 0,Y 331.997,Z 475.759,A -85,B 0,C 180,E1 -14486.359,E2 -14486.359} C_VEL
LIN {X 0,Y 331.917,Z 476.816,A -85,B 0,C 180,E1 -14487.573,E2 -14487.573} C_VEL
LIN {X 0,Y 331.913,Z 477.406,A -85,B 0,C 180,E1 -14488.787,E2 -14488.787} C_VEL
LIN {X 0,Y 331.969,Z 477.561,A -85,B 0,C 180,E1 -14490,E2 -14490} C_VEL
LIN {X 0,Y 331.913,Z 477.406,A -85,B 0,C 180,E1 -14491.213,E2 -14491.213} C_VEL
LIN {X 0,Y 331.917,Z 476.816,A -85,B 0,C 180,E1 -14492.427,E2 -14492.427} C_VEL
LIN {X 0,Y 331.997,Z 475.759,A -85,B 0,C 180,E1 -14493.641,E2 -14493.641} C_VEL
LIN {X 0,Y 332.011,Z 472.997,A -85,B 0,C 180,E1 -14495.787,E2 -14495.787} C_VEL
LIN {X 0,Y 332.362,Z 468.961,A -85,B 0,C 180,E1 -14497.9,E2 -14497.9} C_VEL
LIN {X 0,Y 332.806,Z 464.215,A -85,B 0,C 180,E1 -14499.726,E2 -14499.726} C_VEL
LIN {X 0,Y 333.469,Z 458.19,A -85,B 0,C 180,E1 -14501.55,E2 -14501.55} C_VEL
LIN {X 0,Y 334.314,Z 452.095,A -85,B 0,C 180,E1 -14503.061,E2 -14503.061} C_VEL
LIN {X 0,Y 335.105,Z 446.395,A -85,B 0,C 180,E1 -14504.266,E2 -14504.266} C_VEL
LIN {X 0,Y 336.134,Z 437.838,A -85,B 0,C 180,E1 -14505.772,E2 -14505.772} C_VEL
LIN {X 0,Y 337.083,Z 429.655,A -85,B 0,C 180,E1 -14506.971,E2 -14506.971} C_VEL
LIN {X 0,Y 338.203,Z 421.146,A -85,B 0,C 180,E1 -14508.005,E2 -14508.005} C_VEL
LIN {X 0,Y 339.106,Z 412.428,A -85,B 0,C 180,E1 -14508.895,E2 -14508.895} C_VEL
LIN {X 0,Y 338.192,Z 402.788,A -85,B 0,C 180,E1 -14509.802,E2 -14509.802} C_VEL
LIN {X 0,Y 336.819,Z 393.496,A -85,B 0,C 180,E1 -14510.553,E2 -14510.553} C_VEL
LIN {X 0,Y 334.875,Z 383.251,A -85,B 0,C 180,E1 -14511.247,E2 -14511.247} C_VEL
LIN {X 0,Y 332.486,Z 373.597,A -85,B 0,C 180,E1 -14511.798,E2 -14511.798} C_VEL
LIN {X 0,Y 332.382,Z 372.586,A -85,B 0,C 180,E1 -14511.874,E2 -14511.874} C_VEL
LIN {X 0,Y 332.641,Z 368.83,A -85,B 0,C 180,E1 -14514.996,E2 -14514.996} C_VEL
LIN {X 0,Y 332.949,Z 365.683,A -85,B 0,C 180,E1 -14517.67,E2 -14517.67} C_VEL
LIN {X 0,Y 333.298,Z 362.542,A -85,B 0,C 180,E1 -14520.402,E2 -14520.402} C_VEL
LIN {X 0,Y 333.649,Z 359.429,A -85,B 0,C 180,E1 -14523.207,E2 -14523.207} C_VEL
LIN {X 0,Y 334.17,Z 355.444,A -85,B 0,C 180,E1 -14526.947,E2 -14526.947} C_VEL
LIN {X 0,Y 334.449,Z 353.274,A -85,B 0,C 180,E1 -14529.08,E2 -14529.08} C_VEL
LIN {X 0,Y 334.734,Z 350.231,A -85,B 0,C 180,E1 -14532.211,E2 -14532.211} C_VEL
LIN {X 0,Y 334.625,Z 347.261,A -85,B 0,C 180,E1 -14535.568,E2 -14535.568} C_VEL
LIN {X 0,Y 334.212,Z 344.208,A -85,B 0,C 180,E1 -14539.315,E2 -14539.315} C_VEL
LIN {X 0,Y 333.802,Z 341.441,A -85,B 0,C 180,E1 -14543.136,E2 -14543.136} C_VEL
LIN {X 0,Y 333.675,Z 340.427,A -85,B 0,C 180,E1 -14545.341,E2 -14545.341} C_VEL
LIN {X 0,Y 333.691,Z 340.421,A -85,B 0,C 180,E1 -14549.637,E2 -14549.637} C_VEL
LIN {X 0,Y 333.741,Z 340.411,A -85,B 0,C 180,E1 -14552.4,E2 -14552.4} C_VEL
LIN {X 0,Y 333.726,Z 340.413,A -85,B 0,C 180,E1 -14555.09,E2 -14555.09} C_VEL
LIN {X 0,Y 333.671,Z 340.42,A -85,B 0,C 180,E1 -14559.018,E2 -14559.018} C_VEL
LIN {X 0,Y 333.741,Z 340.416,A -85,B 0,C 180,E1 -14561.586,E2 -14561.586} C_VEL
LIN {X 0,Y 333.808,Z 340.407,A -85,B 0,C 180,E1 -14565.576,E2 -14565.576} C_VEL
LIN {X 0,Y 333.834,Z 340.401,A -85,B 0,C 180,E1 -14569.077,E2 -14569.077} C_VEL
LIN {X 0,Y 334.012,Z 340.377,A -85,B 0,C 180,E1 -14572.747,E2 -14572.747} C_VEL
LIN {X 0,Y 333.808,Z 340.406,A -85,B 0,C 180,E1 -14575.168,E2 -14575.168} C_VEL
LIN {X 0,Y 334.106,Z 340.366,A -85,B 0,C 180,E1 -14577.588,E2 -14577.588} C_VEL
LIN {X 0,Y 334.227,Z 340.347,A -85,B 0,C 180,E1 -14579.999,E2 -14579.999} C_VEL
LIN {X 0,Y 334.106,Z 340.36,A -85,B 0,C 180,E1 -14582.411,E2 -14582.411} C_VEL
LIN {X 0,Y 333.994,Z 340.377,A -85,B 0,C 180,E1 -14586.587,E2 -14586.587} C_VEL
LIN {X 0,Y 333.859,Z 340.394,A -85,B 0,C 180,E1 -14589.694,E2 -14589.694} C_VEL
LIN {X 0,Y 333.795,Z 340.404,A -85,B 0,C 180,E1 -14593.391,E2 -14593.391} C_VEL
LIN {X 0,Y 333.745,Z 340.412,A -85,B 0,C 180,E1 -14597.146,E2 -14597.146} C_VEL
LIN {X 0,Y 333.733,Z 340.41,A -85,B 0,C 180,E1 -14599.69,E2 -14599.69} C_VEL
LIN {X 0,Y 333.667,Z 340.419,A -85,B 0,C 180,E1 -14603.59,E2 -14603.59} C_VEL
LIN {X 0,Y 333.733,Z 340.413,A -85,B 0,C 180,E1 -14606.246,E2 -14606.246} C_VEL
LIN {X 0,Y 333.708,Z 340.415,A -85,B 0,C 180,E1 -14608.971,E2 -14608.971} C_VEL
LIN {X 0,Y 333.643,Z 340.426,A -85,B 0,C 180,E1 -14612.587,E2 -14612.587} C_VEL
LIN {X 0,Y 333.674,Z 340.422,A -85,B 0,C 180,E1 -14616.138,E2 -14616.138} C_VEL
LIN {X 0,Y 333.681,Z 340.417,A -85,B 0,C 180,E1 -14619.187,E2 -14619.187} C_VEL
LIN {X 0,Y 333.688,Z 340.419,A -85,B 0,C 180,E1 -14622.511,E2 -14622.511} C_VEL
LIN {X 0,Y 333.657,Z 340.425,A -85,B 0,C 180,E1 -14625.965,E2 -14625.965} C_VEL
LIN {X 0,Y 333.653,Z 340.421,A -85,B 0,C 180,E1 -14629.313,E2 -14629.313} C_VEL
LIN {X 0,Y 333.652,Z 340.423,A -85,B 0,C 180,E1 -14632.349,E2 -14632.349} C_VEL
LIN {X 0,Y 333.67,Z 340.42,A -85,B 0,C 180,E1 -14635.341,E2 -14635.341} C_VEL
LIN {X 0,Y 333.699,Z 340.421,A -85,B 0,C 180,E1 -14639.71,E2 -14639.71} C_VEL
LIN {X 0,Y 333.739,Z 340.411,A -85,B 0,C 180,E1 -14642.401,E2 -14642.401} C_VEL
LIN {X 0,Y 333.723,Z 340.414,A -85,B 0,C 180,E1 -14645.091,E2 -14645.091} C_VEL
LIN {X 0,Y 333.705,Z 340.463,A -85,B 0,C 180,E1 -14648.779,E2 -14648.779} C_VEL
LIN {X 0,Y 334.601,Z 343.081,A -85,B 0,C 180,E1 -14648.988,E2 -14648.988} C_VEL
LIN {X 0,Y 336.955,Z 345.995,A -85,B 0,C 180,E1 -14649.432,E2 -14649.432} C_VEL
LIN {X 0,Y 339.211,Z 349.263,A -85,B 0,C 180,E1 -14649.878,E2 -14649.878} C_VEL
LIN {X 0,Y 340.701,Z 350.965,A -85,B 0,C 180,E1 -14650.168,E2 -14650.168} C_VEL
LIN {X 0,Y 343.666,Z 354.703,A -85,B 0,C 180,E1 -14650.775,E2 -14650.775} C_VEL
LIN {X 0,Y 345.733,Z 357.177,A -85,B 0,C 180,E1 -14651.206,E2 -14651.206} C_VEL
LIN {X 0,Y 349.02,Z 360.8,A -85,B 0,C 180,E1 -14651.919,E2 -14651.919} C_VEL
LIN {X 0,Y 353.677,Z 366.015,A -85,B 0,C 180,E1 -14652.98,E2 -14652.98} C_VEL
LIN {X 0,Y 356.285,Z 368.571,A -85,B 0,C 180,E1 -14653.603,E2 -14653.603} C_VEL
LIN {X 0,Y 360.088,Z 372.495,A -85,B 0,C 180,E1 -14654.574,E2 -14654.574} C_VEL
LIN {X 0,Y 362.702,Z 374.764,A -85,B 0,C 180,E1 -14655.267,E2 -14655.267} C_VEL
LIN {X 0,Y 366.326,Z 378.564,A -85,B 0,C 180,E1 -14656.341,E2 -14656.341} C_VEL
LIN {X 0,Y 370.092,Z 381.595,A -85,B 0,C 180,E1 -14657.521,E2 -14657.521} C_VEL
LIN {X 0,Y 373.222,Z 384.866,A -85,B 0,C 180,E1 -14658.672,E2 -14658.672} C_VEL
LIN {X 0,Y 376.694,Z 387.408,A -85,B 0,C 180,E1 -14660.003,E2 -14660.003} C_VEL
LIN {X 0,Y 378.714,Z 388.708,A -85,B 0,C 180,E1 -14660.875,E2 -14660.875} C_VEL
LIN {X 0,Y 381.552,Z 392.006,A -85,B 0,C 180,E1 -14662.45,E2 -14662.45} C_VEL
LIN {X 0,Y 384.113,Z 394.036,A -85,B 0,C 180,E1 -14664.093,E2 -14664.093} C_VEL
LIN {X 0,Y 386.261,Z 395.14,A -85,B 0,C 180,E1 -14665.826,E2 -14665.826} C_VEL
LIN {X 0,Y 387.246,Z 395.399,A -85,B 0,C 180,E1 -14666.879,E2 -14666.879} C_VEL
LIN {X 0,Y 387.956,Z 395.547,A -85,B 0,C 180,E1 -14667.924,E2 -14667.924} C_VEL
LIN {X 0,Y 388.401,Z 395.596,A -85,B 0,C 180,E1 -14668.963,E2 -14668.963} C_VEL
LIN {X 0,Y 388.549,Z 395.662,A -85,B 0,C 180,E1 -14670,E2 -14670} C_VEL
LIN {X 0,Y 388.399,Z 395.594,A -85,B 0,C 180,E1 -14671.037,E2 -14671.037} C_VEL
LIN {X 0,Y 387.645,Z 395.501,A -85,B 0,C 180,E1 -14672.598,E2 -14672.598} C_VEL
LIN {X 0,Y 385.632,Z 394.915,A -85,B 0,C 180,E1 -14674.722,E2 -14674.722} C_VEL
LIN {X 0,Y 383.283,Z 393.477,A -85,B 0,C 180,E1 -14676.465,E2 -14676.465} C_VEL
LIN {X 0,Y 380.598,Z 390.976,A -85,B 0,C 180,E1 -14678.102,E2 -14678.102} C_VEL
